LIN {X 0,Y 720.771,Z 351.039,A -85,B 0,C 180,E1 33793.667,E2 33793.667} C_VEL
LIN {X 0,Y 724.023,Z 364.249,A -85,B 0,C 180,E1 33793.246,E2 33793.246} C_VEL
LIN {X 0,Y 722.637,Z 576.137,A -85,B 0,C 180,E1 33790.575,E2 33790.575} C_VEL
LIN {X 0,Y 721.291,Z 800.134,A -85,B 0,C 180,E1 33787.845,E2 33787.845} C_VEL
LIN {X 0,Y 720.97,Z 835.449,A -85,B 0,C 180,E1 33787.381,E2 33787.381} C_VEL
LIN {X 0,Y 720.477,Z 862.842,A -85,B 0,C 180,E1 33786.854,E2 33786.854} C_VEL
LIN {X 0,Y 719.962,Z 888.338,A -85,B 0,C 180,E1 33786.211,E2 33786.211} C_VEL
LIN {X 0,Y 719.265,Z 916.706,A -85,B 0,C 180,E1 33785.311,E2 33785.311} C_VEL
LIN {X 0,Y 718.599,Z 939.502,A -85,B 0,C 180,E1 33784.444,E2 33784.444} C_VEL
LIN {X 0,Y 717.941,Z 960.707,A -85,B 0,C 180,E1 33783.518,E2 33783.518} C_VEL
LIN {X 0,Y 717.25,Z 982.995,A -85,B 0,C 180,E1 33782.412,E2 33782.412} C_VEL
LIN {X 0,Y 716.464,Z 1007.893,A -85,B 0,C 180,E1 33780.994,E2 33780.994} C_VEL
LIN {X 0,Y 715.787,Z 1027.578,A -85,B 0,C 180,E1 33779.728,E2 33779.728} C_VEL
LIN {X 0,Y 715.19,Z 1045.813,A -85,B 0,C 180,E1 33778.431,E2 33778.431} C_VEL
LIN {X 0,Y 714.548,Z 1067.22,A -85,B 0,C 180,E1 33776.735,E2 33776.735} C_VEL
LIN {X 0,Y 713.971,Z 1085.454,A -85,B 0,C 180,E1 33775.108,E2 33775.108} C_VEL
LIN {X 0,Y 713.51,Z 1101.397,A -85,B 0,C 180,E1 33773.539,E2 33773.539} C_VEL
LIN {X 0,Y 713.048,Z 1120.128,A -85,B 0,C 180,E1 33771.468,E2 33771.468} C_VEL
LIN {X 0,Y 712.741,Z 1134.092,A -85,B 0,C 180,E1 33769.723,E2 33769.723} C_VEL
LIN {X 0,Y 712.497,Z 1146.006,A -85,B 0,C 180,E1 33768.067,E2 33768.067} C_VEL
LIN {X 0,Y 712.28,Z 1158.901,A -85,B 0,C 180,E1 33766.054,E2 33766.054} C_VEL
LIN {X 0,Y 712.124,Z 1170.245,A -85,B 0,C 180,E1 33763.975,E2 33763.975} C_VEL
LIN {X 0,Y 712.027,Z 1178.433,A -85,B 0,C 180,E1 33762.242,E2 33762.242} C_VEL
LIN {X 0,Y 711.98,Z 1186.134,A -85,B 0,C 180,E1 33760.355,E2 33760.355} C_VEL
LIN {X 0,Y 711.935,Z 1193.355,A -85,B 0,C 180,E1 33758.155,E2 33758.155} C_VEL
LIN {X 0,Y 711.916,Z 1198.765,A -85,B 0,C 180,E1 33755.966,E2 33755.966} C_VEL
LIN {X 0,Y 711.907,Z 1202.382,A -85,B 0,C 180,E1 33753.866,E2 33753.866} C_VEL
LIN {X 0,Y 711.909,Z 1204.549,A -85,B 0,C 180,E1 33751.61,E2 33751.61} C_VEL
LIN {X 0,Y 711.89,Z 1204.872,A -85,B 0,C 180,E1 33749.517,E2 33749.517} C_VEL
LIN {X 0,Y 711.907,Z 1203.967,A -85,B 0,C 180,E1 33747.585,E2 33747.585} C_VEL
LIN {X 0,Y 711.908,Z 1201.303,A -85,B 0,C 180,E1 33745.408,E2 33745.408} C_VEL
LIN {X 0,Y 711.919,Z 1197.152,A -85,B 0,C 180,E1 33743.306,E2 33743.306} C_VEL
LIN {X 0,Y 711.945,Z 1191.397,A -85,B 0,C 180,E1 33741.195,E2 33741.195} C_VEL
LIN {X 0,Y 711.977,Z 1183.958,A -85,B 0,C 180,E1 33739.071,E2 33739.071} C_VEL
LIN {X 0,Y 712.09,Z 1173.94,A -85,B 0,C 180,E1 33736.769,E2 33736.769} C_VEL
LIN {X 0,Y 712.178,Z 1164.531,A -85,B 0,C 180,E1 33734.946,E2 33734.946} C_VEL
LIN {X 0,Y 712.341,Z 1154.745,A -85,B 0,C 180,E1 33733.277,E2 33733.277} C_VEL
LIN {X 0,Y 712.542,Z 1143.678,A -85,B 0,C 180,E1 33731.595,E2 33731.595} C_VEL
LIN {X 0,Y 712.858,Z 1129.296,A -85,B 0,C 180,E1 33729.644,E2 33729.644} C_VEL
LIN {X 0,Y 713.224,Z 1112.625,A -85,B 0,C 180,E1 33727.672,E2 33727.672} C_VEL
LIN {X 0,Y 713.611,Z 1097.983,A -85,B 0,C 180,E1 33726.114,E2 33726.114} C_VEL
LIN {X 0,Y 714.174,Z 1079.334,A -85,B 0,C 180,E1 33724.317,E2 33724.317} C_VEL
LIN {X 0,Y 714.745,Z 1059.887,A -85,B 0,C 180,E1 33722.665,E2 33722.665} C_VEL
LIN {X 0,Y 715.326,Z 1042.24,A -85,B 0,C 180,E1 33721.306,E2 33721.306} C_VEL
LIN {X 0,Y 716.075,Z 1020.251,A -85,B 0,C 180,E1 33719.777,E2 33719.777} C_VEL
LIN {X 0,Y 716.773,Z 997.046,A -85,B 0,C 180,E1 33718.366,E2 33718.366} C_VEL
LIN {X 0,Y 717.451,Z 976.762,A -85,B 0,C 180,E1 33717.267,E2 33717.267} C_VEL
LIN {X 0,Y 718.191,Z 954.383,A -85,B 0,C 180,E1 33716.192,E2 33716.192} C_VEL
LIN {X 0,Y 718.939,Z 927.69,A -85,B 0,C 180,E1 33715.09,E2 33715.09} C_VEL
LIN {X 0,Y 719.505,Z 905.6,A -85,B 0,C 180,E1 33714.317,E2 33714.317} C_VEL
LIN {X 0,Y 720.071,Z 882.549,A -85,B 0,C 180,E1 33713.63,E2 33713.63} C_VEL
LIN {X 0,Y 720.646,Z 855.599,A -85,B 0,C 180,E1 33712.99,E2 33712.99} C_VEL
LIN {X 0,Y 721.041,Z 828.402,A -85,B 0,C 180,E1 33712.512,E2 33712.512} C_VEL
LIN {X 0,Y 722.489,Z 599.337,A -85,B 0,C 180,E1 33709.712,E2 33709.712} C_VEL
LIN {X 0,Y 723.84,Z 391.194,A -85,B 0,C 180,E1 33707.099,E2 33707.099} C_VEL
LIN {X 0,Y 723.859,Z 362.91,A -85,B 0,C 180,E1 33706.724,E2 33706.724} C_VEL
LIN {X 0,Y 720.673,Z 350.184,A -85,B 0,C 180,E1 33706.291,E2 33706.291} C_VEL
LIN {X 0,Y 720.959,Z 334.838,A -85,B 0,C 180,E1 33705.242,E2 33705.242} C_VEL
LIN {X 0,Y 713.885,Z 319.445,A -85,B 0,C 180,E1 33703.56,E2 33703.56} C_VEL
LIN {X 0,Y 712.33,Z 316.032,A -85,B 0,C 180,E1 33703.177,E2 33703.177} C_VEL
LIN {X 0,Y 712.25,Z 315.511,A -85,B 0,C 180,E1 33703.116,E2 33703.116} C_VEL
LIN {X 0,Y 712.269,Z 315.495,A -85,B 0,C 180,E1 33700.213,E2 33700.213} C_VEL
LIN {X 0,Y 712.243,Z 315.502,A -85,B 0,C 180,E1 33697.335,E2 33697.335} C_VEL
LIN {X 0,Y 712.278,Z 315.499,A -85,B 0,C 180,E1 33694.453,E2 33694.453} C_VEL
LIN {X 0,Y 712.252,Z 315.506,A -85,B 0,C 180,E1 33691.388,E2 33691.388} C_VEL
LIN {X 0,Y 712.258,Z 315.499,A -85,B 0,C 180,E1 33688.506,E2 33688.506} C_VEL
LIN {X 0,Y 712.255,Z 315.499,A -85,B 0,C 180,E1 33685.352,E2 33685.352} C_VEL
LIN {X 0,Y 712.24,Z 315.504,A -85,B 0,C 180,E1 33682.525,E2 33682.525} C_VEL
LIN {X 0,Y 712.279,Z 315.497,A -85,B 0,C 180,E1 33679.518,E2 33679.518} C_VEL
LIN {X 0,Y 712.225,Z 315.505,A -85,B 0,C 180,E1 33676.726,E2 33676.726} C_VEL
LIN {X 0,Y 712.27,Z 315.492,A -85,B 0,C 180,E1 33673.973,E2 33673.973} C_VEL
LIN {X 0,Y 712.235,Z 315.505,A -85,B 0,C 180,E1 33670.925,E2 33670.925} C_VEL
LIN {X 0,Y 712.225,Z 315.498,A -85,B 0,C 180,E1 33668.226,E2 33668.226} C_VEL
LIN {X 0,Y 712.281,Z 315.51,A -85,B 0,C 180,E1 33665.316,E2 33665.316} C_VEL
LIN {X 0,Y 712.213,Z 315.501,A -85,B 0,C 180,E1 33662.494,E2 33662.494} C_VEL
LIN {X 0,Y 712.227,Z 315.506,A -85,B 0,C 180,E1 33659.92,E2 33659.92} C_VEL
LIN {X 0,Y 712.251,Z 315.499,A -85,B 0,C 180,E1 33656.861,E2 33656.861} C_VEL
LIN {X 0,Y 712.205,Z 315.509,A -85,B 0,C 180,E1 33654.198,E2 33654.198} C_VEL
LIN {X 0,Y 712.231,Z 315.5,A -85,B 0,C 180,E1 33651.605,E2 33651.605} C_VEL
LIN {X 0,Y 712.22,Z 315.511,A -85,B 0,C 180,E1 33648.49,E2 33648.49} C_VEL
LIN {X 0,Y 712.196,Z 315.502,A -85,B 0,C 180,E1 33645.953,E2 33645.953} C_VEL
LIN {X 0,Y 712.231,Z 315.503,A -85,B 0,C 180,E1 33643.358,E2 33643.358} C_VEL
LIN {X 0,Y 712.28,Z 315.503,A -85,B 0,C 180,E1 33640.816,E2 33640.816} C_VEL
LIN {X 0,Y 711.26,Z 315.62,A -85,B 0,C 180,E1 33640.197,E2 33640.197} C_VEL
LIN {X 0,Y 704.805,Z 316.435,A -85,B 0,C 180,E1 33638.461,E2 33638.461} C_VEL
LIN {X 0,Y 704.255,Z 316.499,A -85,B 0,C 180,E1 33638.01,E2 33638.01} C_VEL
LIN {X 0,Y 704.249,Z 316.497,A -85,B 0,C 180,E1 33635.596,E2 33635.596} C_VEL
LIN {X 0,Y 704.329,Z 316.492,A -85,B 0,C 180,E1 33632.798,E2 33632.798} C_VEL
LIN {X 0,Y 704.251,Z 316.488,A -85,B 0,C 180,E1 33629.921,E2 33629.921} C_VEL
LIN {X 0,Y 704.239,Z 316.502,A -85,B 0,C 180,E1 33627.495,E2 33627.495} C_VEL
LIN {X 0,Y 704.264,Z 316.488,A -85,B 0,C 180,E1 33624.999,E2 33624.999} C_VEL
LIN {X 0,Y 704.252,Z 316.49,A -85,B 0,C 180,E1 33621.858,E2 33621.858} C_VEL
LIN {X 0,Y 704.231,Z 316.505,A -85,B 0,C 180,E1 33619.427,E2 33619.427} C_VEL
LIN {X 0,Y 704.241,Z 316.504,A -85,B 0,C 180,E1 33617.038,E2 33617.038} C_VEL
LIN {X 0,Y 704.252,Z 316.642,A -85,B 0,C 180,E1 33615.256,E2 33615.256} C_VEL
LIN {X 0,Y 705.594,Z 320.045,A -85,B 0,C 180,E1 33614.883,E2 33614.883} C_VEL
LIN {X 0,Y 706.502,Z 321.785,A -85,B 0,C 180,E1 33614.727,E2 33614.727} C_VEL
LIN {X 0,Y 718.08,Z 339.407,A -85,B 0,C 180,E1 33613.579,E2 33613.579} C_VEL
LIN {X 0,Y 716.627,Z 536.634,A -85,B 0,C 180,E1 33611.066,E2 33611.066} C_VEL
LIN {X 0,Y 715.015,Z 763.363,A -85,B 0,C 180,E1 33608.276,E2 33608.276} C_VEL
LIN {X 0,Y 714.605,Z 804.25,A -85,B 0,C 180,E1 33607.747,E2 33607.747} C_VEL
LIN {X 0,Y 714.056,Z 831.612,A -85,B 0,C 180,E1 33607.225,E2 33607.225} C_VEL
LIN {X 0,Y 713.456,Z 856.532,A -85,B 0,C 180,E1 33606.602,E2 33606.602} C_VEL
LIN {X 0,Y 712.726,Z 883.752,A -85,B 0,C 180,E1 33605.753,E2 33605.753} C_VEL
LIN {X 0,Y 711.881,Z 908.474,A -85,B 0,C 180,E1 33604.816,E2 33604.816} C_VEL
LIN {X 0,Y 711.111,Z 929.791,A -85,B 0,C 180,E1 33603.883,E2 33603.883} C_VEL
LIN {X 0,Y 710.333,Z 950.383,A -85,B 0,C 180,E1 33602.862,E2 33602.862} C_VEL
LIN {X 0,Y 709.442,Z 974.728,A -85,B 0,C 180,E1 33601.494,E2 33601.494} C_VEL
LIN {X 0,Y 708.6,Z 996.129,A -85,B 0,C 180,E1 33600.118,E2 33600.118} C_VEL
LIN {X 0,Y 707.868,Z 1014.676,A -85,B 0,C 180,E1 33598.794,E2 33598.794} C_VEL
LIN {X 0,Y 707.09,Z 1035.698,A -85,B 0,C 180,E1 33597.131,E2 33597.131} C_VEL
LIN {X 0,Y 706.407,Z 1054.988,A -85,B 0,C 180,E1 33595.396,E2 33595.396} C_VEL
LIN {X 0,Y 705.839,Z 1071.299,A -85,B 0,C 180,E1 33593.776,E2 33593.776} C_VEL
LIN {X 0,Y 705.294,Z 1089.764,A -85,B 0,C 180,E1 33591.716,E2 33591.716} C_VEL
LIN {X 0,Y 704.924,Z 1103.476,A -85,B 0,C 180,E1 33589.988,E2 33589.988} C_VEL
LIN {X 0,Y 704.625,Z 1115.703,A -85,B 0,C 180,E1 33588.276,E2 33588.276} C_VEL
LIN {X 0,Y 704.363,Z 1128.113,A -85,B 0,C 180,E1 33586.324,E2 33586.324} C_VEL
LIN {X 0,Y 704.168,Z 1140.163,A -85,B 0,C 180,E1 33584.108,E2 33584.108} C_VEL
LIN {X 0,Y 704.054,Z 1148.655,A -85,B 0,C 180,E1 33582.286,E2 33582.286} C_VEL
LIN {X 0,Y 703.993,Z 1156.268,A -85,B 0,C 180,E1 33580.392,E2 33580.392} C_VEL
LIN {X 0,Y 703.948,Z 1163.465,A -85,B 0,C 180,E1 33578.166,E2 33578.166} C_VEL
LIN {X 0,Y 703.923,Z 1168.842,A -85,B 0,C 180,E1 33575.952,E2 33575.952} C_VEL
LIN {X 0,Y 703.911,Z 1172.427,A -85,B 0,C 180,E1 33573.828,E2 33573.828} C_VEL
LIN {X 0,Y 703.907,Z 1174.519,A -85,B 0,C 180,E1 33571.628,E2 33571.628} C_VEL
LIN {X 0,Y 703.89,Z 1174.884,A -85,B 0,C 180,E1 33569.512,E2 33569.512} C_VEL
LIN {X 0,Y 703.905,Z 1173.934,A -85,B 0,C 180,E1 33567.476,E2 33567.476} C_VEL
LIN {X 0,Y 703.909,Z 1171.247,A -85,B 0,C 180,E1 33565.274,E2 33565.274} C_VEL
LIN {X 0,Y 703.919,Z 1167.064,A -85,B 0,C 180,E1 33563.147,E2 33563.147} C_VEL
LIN {X 0,Y 703.951,Z 1161.278,A -85,B 0,C 180,E1 33561.011,E2 33561.011} C_VEL
LIN {X 0,Y 704.003,Z 1153.813,A -85,B 0,C 180,E1 33558.863,E2 33558.863} C_VEL
LIN {X 0,Y 704.126,Z 1143.751,A -85,B 0,C 180,E1 33556.533,E2 33556.533} C_VEL
LIN {X 0,Y 704.243,Z 1134.314,A -85,B 0,C 180,E1 33554.688,E2 33554.688} C_VEL
LIN {X 0,Y 704.447,Z 1124.499,A -85,B 0,C 180,E1 33552.999,E2 33552.999} C_VEL
LIN {X 0,Y 704.706,Z 1112.819,A -85,B 0,C 180,E1 33551.212,E2 33551.212} C_VEL
LIN {X 0,Y 705.097,Z 1096.881,A -85,B 0,C 180,E1 33549.063,E2 33549.063} C_VEL
LIN {X 0,Y 705.498,Z 1082.171,A -85,B 0,C 180,E1 33547.318,E2 33547.318} C_VEL
LIN {X 0,Y 705.976,Z 1067.563,A -85,B 0,C 180,E1 33545.75,E2 33545.75} C_VEL
LIN {X 0,Y 706.596,Z 1049.287,A -85,B 0,C 180,E1 33543.972,E2 33543.972} C_VEL
LIN {X 0,Y 707.315,Z 1029.605,A -85,B 0,C 180,E1 33542.285,E2 33542.285} C_VEL
LIN {X 0,Y 707.977,Z 1012.225,A -85,B 0,C 180,E1 33540.934,E2 33540.934} C_VEL
LIN {X 0,Y 708.85,Z 989.911,A -85,B 0,C 180,E1 33539.368,E2 33539.368} C_VEL
LIN {X 0,Y 709.707,Z 967.008,A -85,B 0,C 180,E1 33537.966,E2 33537.966} C_VEL
LIN {X 0,Y 710.487,Z 946.818,A -85,B 0,C 180,E1 33536.863,E2 33536.863} C_VEL
LIN {X 0,Y 711.289,Z 925.649,A -85,B 0,C 180,E1 33535.835,E2 33535.835} C_VEL
LIN {X 0,Y 712.17,Z 900.127,A -85,B 0,C 180,E1 33534.758,E2 33534.758} C_VEL
LIN {X 0,Y 712.878,Z 875.711,A -85,B 0,C 180,E1 33533.892,E2 33533.892} C_VEL
LIN {X 0,Y 713.545,Z 852.788,A -85,B 0,C 180,E1 33533.205,E2 33533.205} C_VEL
LIN {X 0,Y 714.206,Z 825.892,A -85,B 0,C 180,E1 33532.561,E2 33532.561} C_VEL
LIN {X 0,Y 714.674,Z 798.761,A -85,B 0,C 180,E1 33532.08,E2 33532.08} C_VEL
LIN {X 0,Y 716.381,Z 570.178,A -85,B 0,C 180,E1 33529.262,E2 33529.262} C_VEL
LIN {X 0,Y 717.934,Z 362.47,A -85,B 0,C 180,E1 33526.632,E2 33526.632} C_VEL
LIN {X 0,Y 717.96,Z 338.909,A -85,B 0,C 180,E1 33526.316,E2 33526.316} C_VEL
LIN {X 0,Y 707.614,Z 323.566,A -85,B 0,C 180,E1 33525.297,E2 33525.297} C_VEL
LIN {X 0,Y 705.936,Z 320.494,A -85,B 0,C 180,E1 33525.089,E2 33525.089} C_VEL
LIN {X 0,Y 704.379,Z 317.274,A -85,B 0,C 180,E1 33524.714,E2 33524.714} C_VEL
LIN {X 0,Y 704.245,Z 316.508,A -85,B 0,C 180,E1 33524.609,E2 33524.609} C_VEL
LIN {X 0,Y 704.277,Z 316.501,A -85,B 0,C 180,E1 33522.055,E2 33522.055} C_VEL
LIN {X 0,Y 704.256,Z 316.504,A -85,B 0,C 180,E1 33518.974,E2 33518.974} C_VEL
LIN {X 0,Y 704.234,Z 316.504,A -85,B 0,C 180,E1 33516.506,E2 33516.506} C_VEL
LIN {X 0,Y 704.241,Z 316.49,A -85,B 0,C 180,E1 33514.113,E2 33514.113} C_VEL
LIN {X 0,Y 704.294,Z 316.489,A -85,B 0,C 180,E1 33511.124,E2 33511.124} C_VEL
LIN {X 0,Y 704.239,Z 316.502,A -85,B 0,C 180,E1 33508.494,E2 33508.494} C_VEL
LIN {X 0,Y 704.24,Z 316.495,A -85,B 0,C 180,E1 33506.113,E2 33506.113} C_VEL
LIN {X 0,Y 704.329,Z 316.499,A -85,B 0,C 180,E1 33503.296,E2 33503.296} C_VEL
LIN {X 0,Y 704.254,Z 316.485,A -85,B 0,C 180,E1 33500.442,E2 33500.442} C_VEL
LIN {X 0,Y 704.251,Z 316.499,A -85,B 0,C 180,E1 33497.968,E2 33497.968} C_VEL
LIN {X 0,Y 704.319,Z 316.487,A -85,B 0,C 180,E1 33495.227,E2 33495.227} C_VEL
LIN {X 0,Y 704.268,Z 316.498,A -85,B 0,C 180,E1 33492.296,E2 33492.296} C_VEL
LIN {X 0,Y 704.257,Z 316.493,A -85,B 0,C 180,E1 33489.81,E2 33489.81} C_VEL
LIN {X 0,Y 704.32,Z 316.492,A -85,B 0,C 180,E1 33487.095,E2 33487.095} C_VEL
LIN {X 0,Y 704.279,Z 316.49,A -85,B 0,C 180,E1 33484.152,E2 33484.152} C_VEL
LIN {X 0,Y 704.269,Z 316.489,A -85,B 0,C 180,E1 33481.546,E2 33481.546} C_VEL
LIN {X 0,Y 704.344,Z 316.492,A -85,B 0,C 180,E1 33478.698,E2 33478.698} C_VEL
LIN {X 0,Y 704.276,Z 316.487,A -85,B 0,C 180,E1 33475.766,E2 33475.766} C_VEL
LIN {X 0,Y 704.29,Z 316.499,A -85,B 0,C 180,E1 33473.151,E2 33473.151} C_VEL
LIN {X 0,Y 704.326,Z 316.485,A -85,B 0,C 180,E1 33470.109,E2 33470.109} C_VEL
LIN {X 0,Y 704.28,Z 316.496,A -85,B 0,C 180,E1 33467.371,E2 33467.371} C_VEL
LIN {X 0,Y 704.343,Z 316.484,A -85,B 0,C 180,E1 33464.521,E2 33464.521} C_VEL
LIN {X 0,Y 704.294,Z 316.493,A -85,B 0,C 180,E1 33461.543,E2 33461.543} C_VEL
LIN {X 0,Y 704.308,Z 316.486,A -85,B 0,C 180,E1 33458.776,E2 33458.776} C_VEL
LIN {X 0,Y 704.326,Z 316.483,A -85,B 0,C 180,E1 33455.688,E2 33455.688} C_VEL
LIN {X 0,Y 704.297,Z 316.495,A -85,B 0,C 180,E1 33452.888,E2 33452.888} C_VEL
LIN {X 0,Y 704.338,Z 316.485,A -85,B 0,C 180,E1 33449.99,E2 33449.99} C_VEL
LIN {X 0,Y 704.3,Z 316.493,A -85,B 0,C 180,E1 33447.061,E2 33447.061} C_VEL
LIN {X 0,Y 704.34,Z 316.498,A -85,B 0,C 180,E1 33444.152,E2 33444.152} C_VEL
LIN {X 0,Y 704.317,Z 316.495,A -85,B 0,C 180,E1 33441.135,E2 33441.135} C_VEL
LIN {X 0,Y 704.339,Z 316.499,A -85,B 0,C 180,E1 33438.147,E2 33438.147} C_VEL
LIN {X 0,Y 704.354,Z 316.627,A -85,B 0,C 180,E1 33437.474,E2 33437.474} C_VEL
LIN {X 0,Y 705.691,Z 320.07,A -85,B 0,C 180,E1 33437.097,E2 33437.097} C_VEL
LIN {X 0,Y 712.541,Z 334.723,A -85,B 0,C 180,E1 33435.441,E2 33435.441} C_VEL
LIN {X 0,Y 714.569,Z 339.653,A -85,B 0,C 180,E1 33434.924,E2 33434.924} C_VEL
LIN {X 0,Y 714.39,Z 351.16,A -85,B 0,C 180,E1 33434.156,E2 33434.156} C_VEL
LIN {X 0,Y 718.167,Z 366.394,A -85,B 0,C 180,E1 33433.658,E2 33433.658} C_VEL
LIN {X 0,Y 716.542,Z 577.372,A -85,B 0,C 180,E1 33430.977,E2 33430.977} C_VEL
LIN {X 0,Y 714.958,Z 801.305,A -85,B 0,C 180,E1 33428.225,E2 33428.225} C_VEL
LIN {X 0,Y 714.581,Z 835.878,A -85,B 0,C 180,E1 33427.766,E2 33427.766} C_VEL
LIN {X 0,Y 714.012,Z 863.03,A -85,B 0,C 180,E1 33427.239,E2 33427.239} C_VEL
LIN {X 0,Y 713.419,Z 888.317,A -85,B 0,C 180,E1 33426.597,E2 33426.597} C_VEL
LIN {X 0,Y 712.6,Z 916.851,A -85,B 0,C 180,E1 33425.686,E2 33425.686} C_VEL
LIN {X 0,Y 711.838,Z 939.505,A -85,B 0,C 180,E1 33424.818,E2 33424.818} C_VEL
LIN {X 0,Y 711.114,Z 959.717,A -85,B 0,C 180,E1 33423.931,E2 33423.931} C_VEL
LIN {X 0,Y 710.335,Z 980.327,A -85,B 0,C 180,E1 33422.91,E2 33422.91} C_VEL
LIN {X 0,Y 709.435,Z 1004.952,A -85,B 0,C 180,E1 33421.525,E2 33421.525} C_VEL
LIN {X 0,Y 708.563,Z 1026.865,A -85,B 0,C 180,E1 33420.113,E2 33420.113} C_VEL
LIN {X 0,Y 707.854,Z 1045.266,A -85,B 0,C 180,E1 33418.794,E2 33418.794} C_VEL
LIN {X 0,Y 707.076,Z 1066.205,A -85,B 0,C 180,E1 33417.132,E2 33417.132} C_VEL
LIN {X 0,Y 706.405,Z 1085.046,A -85,B 0,C 180,E1 33415.435,E2 33415.435} C_VEL
LIN {X 0,Y 705.831,Z 1101.399,A -85,B 0,C 180,E1 33413.811,E2 33413.811} C_VEL
LIN {X 0,Y 705.276,Z 1120.13,A -85,B 0,C 180,E1 33411.716,E2 33411.716} C_VEL
LIN {X 0,Y 704.918,Z 1133.811,A -85,B 0,C 180,E1 33409.989,E2 33409.989} C_VEL
LIN {X 0,Y 704.607,Z 1146.59,A -85,B 0,C 180,E1 33408.191,E2 33408.191} C_VEL
LIN {X 0,Y 704.335,Z 1160.068,A -85,B 0,C 180,E1 33406.036,E2 33406.036} C_VEL
LIN {X 0,Y 704.164,Z 1170.657,A -85,B 0,C 180,E1 33404.052,E2 33404.052} C_VEL
LIN {X 0,Y 704.053,Z 1178.792,A -85,B 0,C 180,E1 33402.299,E2 33402.299} C_VEL
LIN {X 0,Y 703.99,Z 1186.427,A -85,B 0,C 180,E1 33400.392,E2 33400.392} C_VEL
LIN {X 0,Y 703.94,Z 1193.595,A -85,B 0,C 180,E1 33398.166,E2 33398.166} C_VEL
LIN {X 0,Y 703.918,Z 1198.937,A -85,B 0,C 180,E1 33395.952,E2 33395.952} C_VEL
LIN {X 0,Y 703.908,Z 1202.484,A -85,B 0,C 180,E1 33393.828,E2 33393.828} C_VEL
LIN {X 0,Y 703.908,Z 1204.549,A -85,B 0,C 180,E1 33391.628,E2 33391.628} C_VEL
LIN {X 0,Y 703.89,Z 1204.872,A -85,B 0,C 180,E1 33389.512,E2 33389.512} C_VEL
LIN {X 0,Y 703.907,Z 1203.964,A -85,B 0,C 180,E1 33387.558,E2 33387.558} C_VEL
LIN {X 0,Y 703.909,Z 1201.428,A -85,B 0,C 180,E1 33385.438,E2 33385.438} C_VEL
LIN {X 0,Y 703.921,Z 1197.348,A -85,B 0,C 180,E1 33383.311,E2 33383.311} C_VEL
LIN {X 0,Y 703.949,Z 1191.394,A -85,B 0,C 180,E1 33381.094,E2 33381.094} C_VEL
LIN {X 0,Y 703.992,Z 1184.277,A -85,B 0,C 180,E1 33379.029,E2 33379.029} C_VEL
LIN {X 0,Y 704.128,Z 1173.941,A -85,B 0,C 180,E1 33376.617,E2 33376.617} C_VEL
LIN {X 0,Y 704.237,Z 1164.533,A -85,B 0,C 180,E1 33374.772,E2 33374.772} C_VEL
LIN {X 0,Y 704.437,Z 1154.7,A -85,B 0,C 180,E1 33373.076,E2 33373.076} C_VEL
LIN {X 0,Y 704.667,Z 1143.68,A -85,B 0,C 180,E1 33371.382,E2 33371.382} C_VEL
LIN {X 0,Y 705.06,Z 1128.62,A -85,B 0,C 180,E1 33369.322,E2 33369.322} C_VEL
LIN {X 0,Y 705.487,Z 1112.627,A -85,B 0,C 180,E1 33367.414,E2 33367.414} C_VEL
LIN {X 0,Y 705.974,Z 1097.61,A -85,B 0,C 180,E1 33365.8,E2 33365.8} C_VEL
LIN {X 0,Y 706.607,Z 1078.762,A -85,B 0,C 180,E1 33363.97,E2 33363.97} C_VEL
LIN {X 0,Y 707.314,Z 1059.614,A -85,B 0,C 180,E1 33362.331,E2 33362.331} C_VEL
LIN {X 0,Y 707.955,Z 1042.846,A -85,B 0,C 180,E1 33361.025,E2 33361.025} C_VEL
LIN {X 0,Y 708.73,Z 1022.922,A -85,B 0,C 180,E1 33359.618,E2 33359.618} C_VEL
LIN {X 0,Y 709.633,Z 998.654,A -85,B 0,C 180,E1 33358.105,E2 33358.105} C_VEL
LIN {X 0,Y 710.413,Z 978.546,A -85,B 0,C 180,E1 33356.998,E2 33356.998} C_VEL
LIN {X 0,Y 711.154,Z 958.824,A -85,B 0,C 180,E1 33356.027,E2 33356.027} C_VEL
LIN {X 0,Y 711.932,Z 937.251,A -85,B 0,C 180,E1 33355.089,E2 33355.089} C_VEL
LIN {X 0,Y 712.777,Z 911.467,A -85,B 0,C 180,E1 33354.126,E2 33354.126} C_VEL
LIN {X 0,Y 713.471,Z 885.657,A -85,B 0,C 180,E1 33353.329,E2 33353.329} C_VEL
LIN {X 0,Y 714.088,Z 860.466,A -85,B 0,C 180,E1 33352.705,E2 33352.705} C_VEL
LIN {X 0,Y 714.616,Z 832.883,A -85,B 0,C 180,E1 33352.187,E2 33352.187} C_VEL
LIN {X 0,Y 715.061,Z 786.137,A -85,B 0,C 180,E1 33351.591,E2 33351.591} C_VEL
LIN {X 0,Y 716.677,Z 560.284,A -85,B 0,C 180,E1 33348.809,E2 33348.809} C_VEL
LIN {X 0,Y 718.112,Z 365.493,A -85,B 0,C 180,E1 33346.326,E2 33346.326} C_VEL
LIN {X 0,Y 714.26,Z 350.268,A -85,B 0,C 180,E1 33345.803,E2 33345.803} C_VEL
LIN {X 0,Y 714.571,Z 339.143,A -85,B 0,C 180,E1 33345.04,E2 33345.04} C_VEL
LIN {X 0,Y 707.611,Z 324.147,A -85,B 0,C 180,E1 33343.373,E2 33343.373} C_VEL
LIN {X 0,Y 705.51,Z 319.793,A -85,B 0,C 180,E1 33342.866,E2 33342.866} C_VEL
LIN {X 0,Y 704.337,Z 316.498,A -85,B 0,C 180,E1 33342.512,E2 33342.512} C_VEL
LIN {X 0,Y 704.314,Z 316.501,A -85,B 0,C 180,E1 33339.495,E2 33339.495} C_VEL
LIN {X 0,Y 704.337,Z 316.487,A -85,B 0,C 180,E1 33336.537,E2 33336.537} C_VEL
LIN {X 0,Y 704.313,Z 316.49,A -85,B 0,C 180,E1 33333.424,E2 33333.424} C_VEL
LIN {X 0,Y 704.328,Z 316.487,A -85,B 0,C 180,E1 33330.493,E2 33330.493} C_VEL
LIN {X 0,Y 704.318,Z 316.498,A -85,B 0,C 180,E1 33327.385,E2 33327.385} C_VEL
LIN {X 0,Y 704.309,Z 316.484,A -85,B 0,C 180,E1 33324.491,E2 33324.491} C_VEL
LIN {X 0,Y 704.33,Z 316.488,A -85,B 0,C 180,E1 33321.398,E2 33321.398} C_VEL
LIN {X 0,Y 704.292,Z 316.493,A -85,B 0,C 180,E1 33318.543,E2 33318.543} C_VEL
LIN {X 0,Y 704.342,Z 316.488,A -85,B 0,C 180,E1 33315.648,E2 33315.648} C_VEL
LIN {X 0,Y 704.287,Z 316.497,A -85,B 0,C 180,E1 33312.758,E2 33312.758} C_VEL
LIN {X 0,Y 704.317,Z 316.487,A -85,B 0,C 180,E1 33309.974,E2 33309.974} C_VEL
LIN {X 0,Y 704.303,Z 316.5,A -85,B 0,C 180,E1 33306.931,E2 33306.931} C_VEL
LIN {X 0,Y 704.279,Z 316.489,A -85,B 0,C 180,E1 33304.234,E2 33304.234} C_VEL
LIN {X 0,Y 704.345,Z 316.489,A -85,B 0,C 180,E1 33301.302,E2 33301.302} C_VEL
LIN {X 0,Y 704.275,Z 316.491,A -85,B 0,C 180,E1 33298.454,E2 33298.454} C_VEL
LIN {X 0,Y 704.281,Z 316.488,A -85,B 0,C 180,E1 33295.848,E2 33295.848} C_VEL
LIN {X 0,Y 704.316,Z 316.493,A -85,B 0,C 180,E1 33292.823,E2 33292.823} C_VEL
LIN {X 0,Y 704.263,Z 316.491,A -85,B 0,C 180,E1 33290.158,E2 33290.158} C_VEL
LIN {X 0,Y 704.279,Z 316.497,A -85,B 0,C 180,E1 33287.619,E2 33287.619} C_VEL
LIN {X 0,Y 704.292,Z 316.492,A -85,B 0,C 180,E1 33284.52,E2 33284.52} C_VEL
LIN {X 0,Y 704.255,Z 316.499,A -85,B 0,C 180,E1 33281.97,E2 33281.97} C_VEL
LIN {X 0,Y 704.264,Z 316.485,A -85,B 0,C 180,E1 33279.471,E2 33279.471} C_VEL
LIN {X 0,Y 704.255,Z 316.499,A -85,B 0,C 180,E1 33278.01,E2 33278.01} C_VEL
LIN {X 0,Y 703.238,Z 316.628,A -85,B 0,C 180,E1 33277.383,E2 33277.383} C_VEL
LIN {X 0,Y 696.828,Z 317.423,A -85,B 0,C 180,E1 33275.627,E2 33275.627} C_VEL
LIN {X 0,Y 696.343,Z 317.485,A -85,B 0,C 180,E1 33275.171,E2 33275.171} C_VEL
LIN {X 0,Y 696.325,Z 317.491,A -85,B 0,C 180,E1 33272.087,E2 33272.087} C_VEL
LIN {X 0,Y 696.302,Z 317.475,A -85,B 0,C 180,E1 33269.637,E2 33269.637} C_VEL
LIN {X 0,Y 696.321,Z 317.491,A -85,B 0,C 180,E1 33267.126,E2 33267.126} C_VEL
LIN {X 0,Y 696.32,Z 317.494,A -85,B 0,C 180,E1 33263.942,E2 33263.942} C_VEL
LIN {X 0,Y 696.292,Z 317.478,A -85,B 0,C 180,E1 33261.447,E2 33261.447} C_VEL
LIN {X 0,Y 696.308,Z 317.494,A -85,B 0,C 180,E1 33258.985,E2 33258.985} C_VEL
LIN {X 0,Y 696.346,Z 317.495,A -85,B 0,C 180,E1 33255.974,E2 33255.974} C_VEL
LIN {X 0,Y 696.371,Z 317.803,A -85,B 0,C 180,E1 33255.823,E2 33255.823} C_VEL
LIN {X 0,Y 697.895,Z 321.383,A -85,B 0,C 180,E1 33255.438,E2 33255.438} C_VEL
LIN {X 0,Y 701.49,Z 326.53,A -85,B 0,C 180,E1 33255.067,E2 33255.067} C_VEL
LIN {X 0,Y 712.247,Z 343.156,A -85,B 0,C 180,E1 33253.976,E2 33253.976} C_VEL
LIN {X 0,Y 710.567,Z 539.356,A -85,B 0,C 180,E1 33251.458,E2 33251.458} C_VEL
LIN {X 0,Y 708.714,Z 765.576,A -85,B 0,C 180,E1 33248.652,E2 33248.652} C_VEL
LIN {X 0,Y 708.255,Z 804.915,A -85,B 0,C 180,E1 33248.136,E2 33248.136} C_VEL
LIN {X 0,Y 707.62,Z 832.271,A -85,B 0,C 180,E1 33247.606,E2 33247.606} C_VEL
LIN {X 0,Y 706.937,Z 856.943,A -85,B 0,C 180,E1 33246.983,E2 33246.983} C_VEL
LIN {X 0,Y 706.108,Z 883.765,A -85,B 0,C 180,E1 33246.141,E2 33246.141} C_VEL
LIN {X 0,Y 705.151,Z 908.485,A -85,B 0,C 180,E1 33245.197,E2 33245.197} C_VEL
LIN {X 0,Y 704.3,Z 929.261,A -85,B 0,C 180,E1 33244.283,E2 33244.283} C_VEL
LIN {X 0,Y 703.426,Z 949.507,A -85,B 0,C 180,E1 33243.275,E2 33243.275} C_VEL
LIN {X 0,Y 702.397,Z 972.99,A -85,B 0,C 180,E1 33241.958,E2 33241.958} C_VEL
LIN {X 0,Y 701.393,Z 995.625,A -85,B 0,C 180,E1 33240.497,E2 33240.497} C_VEL
LIN {X 0,Y 700.56,Z 1014.141,A -85,B 0,C 180,E1 33239.165,E2 33239.165} C_VEL
LIN {X 0,Y 699.716,Z 1033.482,A -85,B 0,C 180,E1 33237.627,E2 33237.627} C_VEL
LIN {X 0,Y 698.891,Z 1053.297,A -85,B 0,C 180,E1 33235.855,E2 33235.855} C_VEL
LIN {X 0,Y 698.263,Z 1069.266,A -85,B 0,C 180,E1 33234.265,E2 33234.265} C_VEL
LIN {X 0,Y 697.658,Z 1086.03,A -85,B 0,C 180,E1 33232.418,E2 33232.418} C_VEL
LIN {X 0,Y 697.129,Z 1102.193,A -85,B 0,C 180,E1 33230.397,E2 33230.397} C_VEL
LIN {X 0,Y 696.79,Z 1114.544,A -85,B 0,C 180,E1 33228.662,E2 33228.662} C_VEL
LIN {X 0,Y 696.504,Z 1126.043,A -85,B 0,C 180,E1 33226.857,E2 33226.857} C_VEL
LIN {X 0,Y 696.267,Z 1138.389,A -85,B 0,C 180,E1 33224.64,E2 33224.64} C_VEL
LIN {X 0,Y 696.102,Z 1148.244,A -85,B 0,C 180,E1 33222.526,E2 33222.526} C_VEL
LIN {X 0,Y 695.996,Z 1155.965,A -85,B 0,C 180,E1 33220.596,E2 33220.596} C_VEL
LIN {X 0,Y 695.957,Z 1163.223,A -85,B 0,C 180,E1 33218.343,E2 33218.343} C_VEL
LIN {X 0,Y 695.927,Z 1168.672,A -85,B 0,C 180,E1 33216.103,E2 33216.103} C_VEL
LIN {X 0,Y 695.915,Z 1172.318,A -85,B 0,C 180,E1 33213.954,E2 33213.954} C_VEL
LIN {X 0,Y 695.906,Z 1174.463,A -85,B 0,C 180,E1 33211.729,E2 33211.729} C_VEL
LIN {X 0,Y 695.89,Z 1174.884,A -85,B 0,C 180,E1 33209.506,E2 33209.506} C_VEL
LIN {X 0,Y 695.907,Z 1173.999,A -85,B 0,C 180,E1 33207.53,E2 33207.53} C_VEL
LIN {X 0,Y 695.908,Z 1171.496,A -85,B 0,C 180,E1 33205.385,E2 33205.385} C_VEL
LIN {X 0,Y 695.922,Z 1167.454,A -85,B 0,C 180,E1 33203.234,E2 33203.234} C_VEL
LIN {X 0,Y 695.957,Z 1161.528,A -85,B 0,C 180,E1 33200.991,E2 33200.991} C_VEL
LIN {X 0,Y 696.015,Z 1154.336,A -85,B 0,C 180,E1 33198.872,E2 33198.872} C_VEL
LIN {X 0,Y 696.159,Z 1144.155,A -85,B 0,C 180,E1 33196.461,E2 33196.461} C_VEL
LIN {X 0,Y 696.301,Z 1134.778,A -85,B 0,C 180,E1 33194.594,E2 33194.594} C_VEL
LIN {X 0,Y 696.535,Z 1124.497,A -85,B 0,C 180,E1 33192.8,E2 33192.8} C_VEL
LIN {X 0,Y 696.842,Z 1112.817,A -85,B 0,C 180,E1 33190.992,E2 33190.992} C_VEL
LIN {X 0,Y 697.304,Z 1096.874,A -85,B 0,C 180,E1 33188.818,E2 33188.818} C_VEL
LIN {X 0,Y 697.776,Z 1082.243,A -85,B 0,C 180,E1 33187.061,E2 33187.061} C_VEL
LIN {X 0,Y 698.365,Z 1066.705,A -85,B 0,C 180,E1 33185.378,E2 33185.378} C_VEL
LIN {X 0,Y 699.173,Z 1046.349,A -85,B 0,C 180,E1 33183.41,E2 33183.41} C_VEL
LIN {X 0,Y 699.913,Z 1029.044,A -85,B 0,C 180,E1 33181.92,E2 33181.92} C_VEL
LIN {X 0,Y 700.688,Z 1011.093,A -85,B 0,C 180,E1 33180.515,E2 33180.515} C_VEL
LIN {X 0,Y 701.705,Z 988.261,A -85,B 0,C 180,E1 33178.914,E2 33178.914} C_VEL
LIN {X 0,Y 702.664,Z 967.001,A -85,B 0,C 180,E1 33177.606,E2 33177.606} C_VEL
LIN {X 0,Y 703.516,Z 947.591,A -85,B 0,C 180,E1 33176.534,E2 33176.534} C_VEL
LIN {X 0,Y 704.393,Z 927.29,A -85,B 0,C 180,E1 33175.535,E2 33175.535} C_VEL
LIN {X 0,Y 705.424,Z 902.137,A -85,B 0,C 180,E1 33174.45,E2 33174.45} C_VEL
LIN {X 0,Y 706.281,Z 876.183,A -85,B 0,C 180,E1 33173.517,E2 33173.517} C_VEL
LIN {X 0,Y 707.044,Z 853.194,A -85,B 0,C 180,E1 33172.824,E2 33172.824} C_VEL
LIN {X 0,Y 707.777,Z 826.912,A -85,B 0,C 180,E1 33172.186,E2 33172.186} C_VEL
LIN {X 0,Y 708.336,Z 799.401,A -85,B 0,C 180,E1 33171.69,E2 33171.69} C_VEL
LIN {X 0,Y 710.27,Z 574.638,A -85,B 0,C 180,E1 33168.896,E2 33168.896} C_VEL
LIN {X 0,Y 712.082,Z 365.35,A -85,B 0,C 180,E1 33166.225,E2 33166.225} C_VEL
LIN {X 0,Y 712.135,Z 342.734,A -85,B 0,C 180,E1 33165.92,E2 33165.92} C_VEL
LIN {X 0,Y 701.027,Z 326.024,A -85,B 0,C 180,E1 33164.798,E2 33164.798} C_VEL
LIN {X 0,Y 697.409,Z 320.649,A -85,B 0,C 180,E1 33164.4,E2 33164.4} C_VEL
LIN {X 0,Y 696.348,Z 317.495,A -85,B 0,C 180,E1 33164.045,E2 33164.045} C_VEL
LIN {X 0,Y 696.32,Z 317.495,A -85,B 0,C 180,E1 33161.014,E2 33161.014} C_VEL
LIN {X 0,Y 696.297,Z 317.494,A -85,B 0,C 180,E1 33158.553,E2 33158.553} C_VEL
LIN {X 0,Y 696.316,Z 317.493,A -85,B 0,C 180,E1 33156.058,E2 33156.058} C_VEL
LIN {X 0,Y 696.315,Z 317.493,A -85,B 0,C 180,E1 33152.875,E2 33152.875} C_VEL
LIN {X 0,Y 696.295,Z 317.477,A -85,B 0,C 180,E1 33150.459,E2 33150.459} C_VEL
LIN {X 0,Y 696.303,Z 317.491,A -85,B 0,C 180,E1 33148.1,E2 33148.1} C_VEL
LIN {X 0,Y 696.394,Z 317.472,A -85,B 0,C 180,E1 33145.24,E2 33145.24} C_VEL
LIN {X 0,Y 696.308,Z 317.489,A -85,B 0,C 180,E1 33142.367,E2 33142.367} C_VEL
LIN {X 0,Y 696.307,Z 317.473,A -85,B 0,C 180,E1 33139.985,E2 33139.985} C_VEL
LIN {X 0,Y 696.391,Z 317.489,A -85,B 0,C 180,E1 33137.204,E2 33137.204} C_VEL
LIN {X 0,Y 696.319,Z 317.476,A -85,B 0,C 180,E1 33134.248,E2 33134.248} C_VEL
LIN {X 0,Y 696.319,Z 317.489,A -85,B 0,C 180,E1 33131.766,E2 33131.766} C_VEL
LIN {X 0,Y 696.402,Z 317.468,A -85,B 0,C 180,E1 33128.921,E2 33128.921} C_VEL
LIN {X 0,Y 696.327,Z 317.487,A -85,B 0,C 180,E1 33126.017,E2 33126.017} C_VEL
LIN {X 0,Y 696.334,Z 317.481,A -85,B 0,C 180,E1 33123.458,E2 33123.458} C_VEL
LIN {X 0,Y 696.402,Z 317.483,A -85,B 0,C 180,E1 33120.494,E2 33120.494} C_VEL
LIN {X 0,Y 696.332,Z 317.478,A -85,B 0,C 180,E1 33117.696,E2 33117.696} C_VEL
LIN {X 0,Y 696.371,Z 317.479,A -85,B 0,C 180,E1 33114.975,E2 33114.975} C_VEL
LIN {X 0,Y 696.356,Z 317.475,A -85,B 0,C 180,E1 33111.911,E2 33111.911} C_VEL
LIN {X 0,Y 696.342,Z 317.479,A -85,B 0,C 180,E1 33109.241,E2 33109.241} C_VEL
LIN {X 0,Y 696.404,Z 317.471,A -85,B 0,C 180,E1 33106.296,E2 33106.296} C_VEL
LIN {X 0,Y 696.346,Z 317.481,A -85,B 0,C 180,E1 33103.396,E2 33103.396} C_VEL
LIN {X 0,Y 696.395,Z 317.474,A -85,B 0,C 180,E1 33100.542,E2 33100.542} C_VEL
LIN {X 0,Y 696.367,Z 317.483,A -85,B 0,C 180,E1 33097.546,E2 33097.546} C_VEL
LIN {X 0,Y 696.365,Z 317.474,A -85,B 0,C 180,E1 33094.757,E2 33094.757} C_VEL
LIN {X 0,Y 696.399,Z 317.476,A -85,B 0,C 180,E1 33091.656,E2 33091.656} C_VEL
LIN {X 0,Y 696.362,Z 317.483,A -85,B 0,C 180,E1 33088.778,E2 33088.778} C_VEL
LIN {X 0,Y 696.397,Z 317.473,A -85,B 0,C 180,E1 33085.847,E2 33085.847} C_VEL
LIN {X 0,Y 696.365,Z 317.479,A -85,B 0,C 180,E1 33082.97,E2 33082.97} C_VEL
LIN {X 0,Y 696.402,Z 317.483,A -85,B 0,C 180,E1 33080.057,E2 33080.057} C_VEL
LIN {X 0,Y 696.418,Z 317.603,A -85,B 0,C 180,E1 33078.115,E2 33078.115} C_VEL
LIN {X 0,Y 697.598,Z 320.815,A -85,B 0,C 180,E1 33077.76,E2 33077.76} C_VEL
LIN {X 0,Y 698.79,Z 323.249,A -85,B 0,C 180,E1 33077.466,E2 33077.466} C_VEL
LIN {X 0,Y 705.986,Z 338.408,A -85,B 0,C 180,E1 33075.714,E2 33075.714} C_VEL
LIN {X 0,Y 708.138,Z 343.431,A -85,B 0,C 180,E1 33075.172,E2 33075.172} C_VEL
LIN {X 0,Y 708.015,Z 351.11,A -85,B 0,C 180,E1 33074.66,E2 33074.66} C_VEL
LIN {X 0,Y 712.348,Z 368.532,A -85,B 0,C 180,E1 33074.077,E2 33074.077} C_VEL
LIN {X 0,Y 710.481,Z 578.791,A -85,B 0,C 180,E1 33071.385,E2 33071.385} C_VEL
LIN {X 0,Y 708.659,Z 802.298,A -85,B 0,C 180,E1 33068.615,E2 33068.615} C_VEL
LIN {X 0,Y 708.224,Z 836.377,A -85,B 0,C 180,E1 33068.156,E2 33068.156} C_VEL
LIN {X 0,Y 707.584,Z 863.297,A -85,B 0,C 180,E1 33067.628,E2 33067.628} C_VEL
LIN {X 0,Y 706.902,Z 888.48,A -85,B 0,C 180,E1 33066.986,E2 33066.986} C_VEL
LIN {X 0,Y 705.969,Z 916.909,A -85,B 0,C 180,E1 33066.071,E2 33066.071} C_VEL
LIN {X 0,Y 705.111,Z 939.393,A -85,B 0,C 180,E1 33065.204,E2 33065.204} C_VEL
LIN {X 0,Y 704.278,Z 959.72,A -85,B 0,C 180,E1 33064.306,E2 33064.306} C_VEL
LIN {X 0,Y 703.407,Z 979.97,A -85,B 0,C 180,E1 33063.296,E2 33063.296} C_VEL
LIN {X 0,Y 702.349,Z 1004.214,A -85,B 0,C 180,E1 33061.929,E2 33061.929} C_VEL
LIN {X 0,Y 701.361,Z 1026.257,A -85,B 0,C 180,E1 33060.498,E2 33060.498} C_VEL
LIN {X 0,Y 700.54,Z 1044.723,A -85,B 0,C 180,E1 33059.166,E2 33059.166} C_VEL
LIN {X 0,Y 699.646,Z 1065.15,A -85,B 0,C 180,E1 33057.536,E2 33057.536} C_VEL
LIN {X 0,Y 698.843,Z 1084.524,A -85,B 0,C 180,E1 33055.782,E2 33055.782} C_VEL
LIN {X 0,Y 698.206,Z 1100.547,A -85,B 0,C 180,E1 33054.177,E2 33054.177} C_VEL
LIN {X 0,Y 697.593,Z 1118.362,A -85,B 0,C 180,E1 33052.189,E2 33052.189} C_VEL
LIN {X 0,Y 697.09,Z 1133.813,A -85,B 0,C 180,E1 33050.223,E2 33050.223} C_VEL
LIN {X 0,Y 696.733,Z 1146.592,A -85,B 0,C 180,E1 33048.404,E2 33048.404} C_VEL
LIN {X 0,Y 696.411,Z 1159.879,A -85,B 0,C 180,E1 33046.258,E2 33046.258} C_VEL
LIN {X 0,Y 696.216,Z 1170.714,A -85,B 0,C 180,E1 33044.205,E2 33044.205} C_VEL
LIN {X 0,Y 696.087,Z 1178.793,A -85,B 0,C 180,E1 33042.442,E2 33042.442} C_VEL
LIN {X 0,Y 695.998,Z 1186.427,A -85,B 0,C 180,E1 33040.512,E2 33040.512} C_VEL
LIN {X 0,Y 695.949,Z 1193.595,A -85,B 0,C 180,E1 33038.26,E2 33038.26} C_VEL
LIN {X 0,Y 695.92,Z 1198.937,A -85,B 0,C 180,E1 33036.02,E2 33036.02} C_VEL
LIN {X 0,Y 695.908,Z 1202.484,A -85,B 0,C 180,E1 33033.872,E2 33033.872} C_VEL
LIN {X 0,Y 695.908,Z 1204.549,A -85,B 0,C 180,E1 33031.647,E2 33031.647} C_VEL
LIN {X 0,Y 695.89,Z 1204.872,A -85,B 0,C 180,E1 33029.506,E2 33029.506} C_VEL
LIN {X 0,Y 695.907,Z 1203.961,A -85,B 0,C 180,E1 33027.53,E2 33027.53} C_VEL
LIN {X 0,Y 695.909,Z 1201.428,A -85,B 0,C 180,E1 33025.385,E2 33025.385} C_VEL
LIN {X 0,Y 695.922,Z 1197.348,A -85,B 0,C 180,E1 33023.234,E2 33023.234} C_VEL
LIN {X 0,Y 695.957,Z 1191.391,A -85,B 0,C 180,E1 33020.991,E2 33020.991} C_VEL
LIN {X 0,Y 696.017,Z 1184.162,A -85,B 0,C 180,E1 33018.871,E2 33018.871} C_VEL
LIN {X 0,Y 696.165,Z 1173.94,A -85,B 0,C 180,E1 33016.461,E2 33016.461} C_VEL
LIN {X 0,Y 696.309,Z 1164.535,A -85,B 0,C 180,E1 33014.595,E2 33014.595} C_VEL
LIN {X 0,Y 696.535,Z 1154.749,A -85,B 0,C 180,E1 33012.886,E2 33012.886} C_VEL
LIN {X 0,Y 696.81,Z 1143.682,A -85,B 0,C 180,E1 33011.164,E2 33011.164} C_VEL
LIN {X 0,Y 697.256,Z 1128.618,A -85,B 0,C 180,E1 33009.08,E2 33009.08} C_VEL
LIN {X 0,Y 697.77,Z 1112.484,A -85,B 0,C 180,E1 33007.133,E2 33007.133} C_VEL
LIN {X 0,Y 698.354,Z 1097.132,A -85,B 0,C 180,E1 33005.468,E2 33005.468} C_VEL
LIN {X 0,Y 699.102,Z 1077.878,A -85,B 0,C 180,E1 33003.59,E2 33003.59} C_VEL
LIN {X 0,Y 699.908,Z 1059.06,A -85,B 0,C 180,E1 33001.966,E2 33001.966} C_VEL
LIN {X 0,Y 700.676,Z 1041.637,A -85,B 0,C 180,E1 33000.601,E2 33000.601} C_VEL
LIN {X 0,Y 701.655,Z 1019.543,A -85,B 0,C 180,E1 32999.041,E2 32999.041} C_VEL
LIN {X 0,Y 702.662,Z 997.051,A -85,B 0,C 180,E1 32997.654,E2 32997.654} C_VEL
LIN {X 0,Y 703.513,Z 977.658,A -85,B 0,C 180,E1 32996.583,E2 32996.583} C_VEL
LIN {X 0,Y 704.372,Z 957.733,A -85,B 0,C 180,E1 32995.6,E2 32995.6} C_VEL
LIN {X 0,Y 705.354,Z 933.855,A -85,B 0,C 180,E1 32994.566,E2 32994.566} C_VEL
LIN {X 0,Y 706.253,Z 907.072,A -85,B 0,C 180,E1 32993.591,E2 32993.591} C_VEL
LIN {X 0,Y 707.026,Z 883.676,A -85,B 0,C 180,E1 32992.881,E2 32992.881} C_VEL
LIN {X 0,Y 707.751,Z 857.861,A -85,B 0,C 180,E1 32992.252,E2 32992.252} C_VEL
LIN {X 0,Y 708.321,Z 830.11,A -85,B 0,C 180,E1 32991.745,E2 32991.745} C_VEL
LIN {X 0,Y 709.322,Z 718.523,A -85,B 0,C 180,E1 32990.357,E2 32990.357} C_VEL
LIN {X 0,Y 711.206,Z 496.443,A -85,B 0,C 180,E1 32987.573,E2 32987.573} C_VEL
LIN {X 0,Y 712.225,Z 367.35,A -85,B 0,C 180,E1 32985.898,E2 32985.898} C_VEL
LIN {X 0,Y 707.901,Z 350.268,A -85,B 0,C 180,E1 32985.301,E2 32985.301} C_VEL
LIN {X 0,Y 708.077,Z 343.13,A -85,B 0,C 180,E1 32984.801,E2 32984.801} C_VEL
LIN {X 0,Y 700.067,Z 325.696,A -85,B 0,C 180,E1 32982.833,E2 32982.833} C_VEL
LIN {X 0,Y 697.597,Z 320.815,A -85,B 0,C 180,E1 32982.24,E2 32982.24} C_VEL
LIN {X 0,Y 696.4,Z 317.48,A -85,B 0,C 180,E1 32981.857,E2 32981.857} C_VEL
LIN {X 0,Y 696.378,Z 317.485,A -85,B 0,C 180,E1 32978.863,E2 32978.863} C_VEL
LIN {X 0,Y 696.401,Z 317.489,A -85,B 0,C 180,E1 32975.759,E2 32975.759} C_VEL
LIN {X 0,Y 696.37,Z 317.48,A -85,B 0,C 180,E1 32972.774,E2 32972.774} C_VEL
LIN {X 0,Y 696.404,Z 317.471,A -85,B 0,C 180,E1 32969.693,E2 32969.693} C_VEL
LIN {X 0,Y 696.358,Z 317.482,A -85,B 0,C 180,E1 32966.8,E2 32966.8} C_VEL
LIN {X 0,Y 696.399,Z 317.475,A -85,B 0,C 180,E1 32963.855,E2 32963.855} C_VEL
LIN {X 0,Y 696.353,Z 317.472,A -85,B 0,C 180,E1 32960.949,E2 32960.949} C_VEL
LIN {X 0,Y 696.393,Z 317.479,A -85,B 0,C 180,E1 32958.067,E2 32958.067} C_VEL
LIN {X 0,Y 696.357,Z 317.472,A -85,B 0,C 180,E1 32954.979,E2 32954.979} C_VEL
LIN {X 0,Y 696.355,Z 317.483,A -85,B 0,C 180,E1 32952.27,E2 32952.27} C_VEL
LIN {X 0,Y 696.396,Z 317.47,A -85,B 0,C 180,E1 32949.254,E2 32949.254} C_VEL
LIN {X 0,Y 696.338,Z 317.486,A -85,B 0,C 180,E1 32946.431,E2 32946.431} C_VEL
LIN {X 0,Y 696.397,Z 317.473,A -85,B 0,C 180,E1 32943.622,E2 32943.622} C_VEL
LIN {X 0,Y 696.347,Z 317.488,A -85,B 0,C 180,E1 32940.658,E2 32940.658} C_VEL
LIN {X 0,Y 696.336,Z 317.477,A -85,B 0,C 180,E1 32938.025,E2 32938.025} C_VEL
LIN {X 0,Y 696.401,Z 317.481,A -85,B 0,C 180,E1 32935.058,E2 32935.058} C_VEL
LIN {X 0,Y 696.328,Z 317.479,A -85,B 0,C 180,E1 32932.209,E2 32932.209} C_VEL
LIN {X 0,Y 696.35,Z 317.477,A -85,B 0,C 180,E1 32929.576,E2 32929.576} C_VEL
LIN {X 0,Y 696.341,Z 317.479,A -85,B 0,C 180,E1 32926.43,E2 32926.43} C_VEL
LIN {X 0,Y 696.317,Z 317.482,A -85,B 0,C 180,E1 32923.869,E2 32923.869} C_VEL
LIN {X 0,Y 696.378,Z 317.486,A -85,B 0,C 180,E1 32921.118,E2 32921.118} C_VEL
LIN {X 0,Y 696.327,Z 317.488,A -85,B 0,C 180,E1 32918.166,E2 32918.166} C_VEL
LIN {X 0,Y 696.309,Z 317.486,A -85,B 0,C 180,E1 32915.752,E2 32915.752} C_VEL
LIN {X 0,Y 696.343,Z 317.485,A -85,B 0,C 180,E1 32915.171,E2 32915.171} C_VEL
LIN {X 0,Y 695.419,Z 317.608,A -85,B 0,C 180,E1 32914.537,E2 32914.537} C_VEL
LIN {X 0,Y 688.891,Z 318.427,A -85,B 0,C 180,E1 32912.716,E2 32912.716} C_VEL
LIN {X 0,Y 688.411,Z 318.48,A -85,B 0,C 180,E1 32912.3,E2 32912.3} C_VEL
LIN {X 0,Y 688.364,Z 318.462,A -85,B 0,C 180,E1 32909.732,E2 32909.732} C_VEL
LIN {X 0,Y 688.37,Z 318.481,A -85,B 0,C 180,E1 32907.292,E2 32907.292} C_VEL
LIN {X 0,Y 688.442,Z 318.467,A -85,B 0,C 180,E1 32904.38,E2 32904.38} C_VEL
LIN {X 0,Y 688.355,Z 318.466,A -85,B 0,C 180,E1 32901.559,E2 32901.559} C_VEL
LIN {X 0,Y 688.358,Z 318.484,A -85,B 0,C 180,E1 32899.18,E2 32899.18} C_VEL
LIN {X 0,Y 688.446,Z 318.561,A -85,B 0,C 180,E1 32896.445,E2 32896.445} C_VEL
LIN {X 0,Y 689.515,Z 321.61,A -85,B 0,C 180,E1 32896.147,E2 32896.147} C_VEL
LIN {X 0,Y 701.237,Z 338.609,A -85,B 0,C 180,E1 32894.916,E2 32894.916} C_VEL
LIN {X 0,Y 706.451,Z 346.771,A -85,B 0,C 180,E1 32894.382,E2 32894.382} C_VEL
LIN {X 0,Y 704.535,Z 542.968,A -85,B 0,C 180,E1 32891.845,E2 32891.845} C_VEL
LIN {X 0,Y 702.427,Z 769.508,A -85,B 0,C 180,E1 32889.013,E2 32889.013} C_VEL
LIN {X 0,Y 701.926,Z 805.799,A -85,B 0,C 180,E1 32888.527,E2 32888.527} C_VEL
LIN {X 0,Y 701.216,Z 832.93,A -85,B 0,C 180,E1 32887.994,E2 32887.994} C_VEL
LIN {X 0,Y 700.448,Z 857.491,A -85,B 0,C 180,E1 32887.368,E2 32887.368} C_VEL
LIN {X 0,Y 699.459,Z 885.064,A -85,B 0,C 180,E1 32886.488,E2 32886.488} C_VEL
LIN {X 0,Y 698.432,Z 908.919,A -85,B 0,C 180,E1 32885.568,E2 32885.568} C_VEL
LIN {X 0,Y 697.518,Z 928.831,A -85,B 0,C 180,E1 32884.686,E2 32884.686} C_VEL
LIN {X 0,Y 696.555,Z 948.632,A -85,B 0,C 180,E1 32883.696,E2 32883.696} C_VEL
LIN {X 0,Y 695.56,Z 968.722,A -85,B 0,C 180,E1 32882.571,E2 32882.571} C_VEL
LIN {X 0,Y 694.273,Z 993.628,A -85,B 0,C 180,E1 32880.988,E2 32880.988} C_VEL
LIN {X 0,Y 693.291,Z 1013.151,A -85,B 0,C 180,E1 32879.579,E2 32879.579} C_VEL
LIN {X 0,Y 692.429,Z 1030.744,A -85,B 0,C 180,E1 32878.176,E2 32878.176} C_VEL
LIN {X 0,Y 691.417,Z 1051.276,A -85,B 0,C 180,E1 32876.356,E2 32876.356} C_VEL
LIN {X 0,Y 690.65,Z 1068.753,A -85,B 0,C 180,E1 32874.606,E2 32874.606} C_VEL
LIN {X 0,Y 689.968,Z 1084.796,A -85,B 0,C 180,E1 32872.826,E2 32872.826} C_VEL
LIN {X 0,Y 689.326,Z 1101.935,A -85,B 0,C 180,E1 32870.675,E2 32870.675} C_VEL
LIN {X 0,Y 688.926,Z 1114.695,A -85,B 0,C 180,E1 32868.862,E2 32868.862} C_VEL
LIN {X 0,Y 688.6,Z 1126.048,A -85,B 0,C 180,E1 32867.056,E2 32867.056} C_VEL
LIN {X 0,Y 688.313,Z 1138.393,A -85,B 0,C 180,E1 32864.813,E2 32864.813} C_VEL
LIN {X 0,Y 688.136,Z 1148.248,A -85,B 0,C 180,E1 32862.674,E2 32862.674} C_VEL
LIN {X 0,Y 688.008,Z 1155.964,A -85,B 0,C 180,E1 32860.72,E2 32860.72} C_VEL
LIN {X 0,Y 687.963,Z 1163.224,A -85,B 0,C 180,E1 32858.441,E2 32858.441} C_VEL
LIN {X 0,Y 687.931,Z 1168.673,A -85,B 0,C 180,E1 32856.174,E2 32856.174} C_VEL
LIN {X 0,Y 687.916,Z 1172.315,A -85,B 0,C 180,E1 32854.001,E2 32854.001} C_VEL
LIN {X 0,Y 687.907,Z 1174.463,A -85,B 0,C 180,E1 32851.749,E2 32851.749} C_VEL
LIN {X 0,Y 687.891,Z 1174.884,A -85,B 0,C 180,E1 32849.5,E2 32849.5} C_VEL
LIN {X 0,Y 687.906,Z 1173.995,A -85,B 0,C 180,E1 32847.501,E2 32847.501} C_VEL
LIN {X 0,Y 687.909,Z 1171.496,A -85,B 0,C 180,E1 32845.331,E2 32845.331} C_VEL
LIN {X 0,Y 687.925,Z 1167.301,A -85,B 0,C 180,E1 32843.09,E2 32843.09} C_VEL
LIN {X 0,Y 687.967,Z 1161.523,A -85,B 0,C 180,E1 32840.885,E2 32840.885} C_VEL
LIN {X 0,Y 688.038,Z 1154.447,A -85,B 0,C 180,E1 32838.771,E2 32838.771} C_VEL
LIN {X 0,Y 688.193,Z 1144.151,A -85,B 0,C 180,E1 32836.301,E2 32836.301} C_VEL
LIN {X 0,Y 688.396,Z 1134.311,A -85,B 0,C 180,E1 32834.327,E2 32834.327} C_VEL
LIN {X 0,Y 688.634,Z 1124.199,A -85,B 0,C 180,E1 32832.547,E2 32832.547} C_VEL
LIN {X 0,Y 689.016,Z 1111.65,A -85,B 0,C 180,E1 32830.591,E2 32830.591} C_VEL
LIN {X 0,Y 689.563,Z 1095.466,A -85,B 0,C 180,E1 32828.389,E2 32828.389} C_VEL
LIN {X 0,Y 690.142,Z 1080.679,A -85,B 0,C 180,E1 32826.612,E2 32826.612} C_VEL
LIN {X 0,Y 690.875,Z 1063.285,A -85,B 0,C 180,E1 32824.727,E2 32824.727} C_VEL
LIN {X 0,Y 691.768,Z 1044.313,A -85,B 0,C 180,E1 32822.917,E2 32822.917} C_VEL
LIN {X 0,Y 692.575,Z 1027.375,A -85,B 0,C 180,E1 32821.454,E2 32821.454} C_VEL
LIN {X 0,Y 693.622,Z 1006.799,A -85,B 0,C 180,E1 32819.848,E2 32819.848} C_VEL
LIN {X 0,Y 694.76,Z 984.404,A -85,B 0,C 180,E1 32818.313,E2 32818.313} C_VEL
LIN {X 0,Y 695.729,Z 965.387,A -85,B 0,C 180,E1 32817.145,E2 32817.145} C_VEL
LIN {X 0,Y 696.702,Z 945.796,A -85,B 0,C 180,E1 32816.064,E2 32816.064} C_VEL
LIN {X 0,Y 697.769,Z 923.605,A -85,B 0,C 180,E1 32814.978,E2 32814.978} C_VEL
LIN {X 0,Y 698.879,Z 897.557,A -85,B 0,C 180,E1 32813.883,E2 32813.883} C_VEL
LIN {X 0,Y 699.795,Z 874.701,A -85,B 0,C 180,E1 32813.073,E2 32813.073} C_VEL
LIN {X 0,Y 700.639,Z 851.889,A -85,B 0,C 180,E1 32812.388,E2 32812.388} C_VEL
LIN {X 0,Y 701.47,Z 824.908,A -85,B 0,C 180,E1 32811.738,E2 32811.738} C_VEL
LIN {X 0,Y 702.071,Z 797.503,A -85,B 0,C 180,E1 32811.257,E2 32811.257} C_VEL
LIN {X 0,Y 704.257,Z 571.862,A -85,B 0,C 180,E1 32808.431,E2 32808.431} C_VEL
LIN {X 0,Y 706.302,Z 363.947,A -85,B 0,C 180,E1 32805.756,E2 32805.756} C_VEL
LIN {X 0,Y 706.276,Z 346.312,A -85,B 0,C 180,E1 32805.508,E2 32805.508} C_VEL
LIN {X 0,Y 696.491,Z 331.654,A -85,B 0,C 180,E1 32804.503,E2 32804.503} C_VEL
LIN {X 0,Y 689.053,Z 320.664,A -85,B 0,C 180,E1 32803.688,E2 32803.688} C_VEL
LIN {X 0,Y 688.431,Z 318.481,A -85,B 0,C 180,E1 32803.433,E2 32803.433} C_VEL
LIN {X 0,Y 688.364,Z 318.484,A -85,B 0,C 180,E1 32800.708,E2 32800.708} C_VEL
LIN {X 0,Y 688.364,Z 318.483,A -85,B 0,C 180,E1 32798.334,E2 32798.334} C_VEL
LIN {X 0,Y 688.447,Z 318.463,A -85,B 0,C 180,E1 32795.416,E2 32795.416} C_VEL
LIN {X 0,Y 688.357,Z 318.482,A -85,B 0,C 180,E1 32792.599,E2 32792.599} C_VEL
LIN {X 0,Y 688.358,Z 318.464,A -85,B 0,C 180,E1 32790.172,E2 32790.172} C_VEL
LIN {X 0,Y 688.453,Z 318.473,A -85,B 0,C 180,E1 32787.32,E2 32787.32} C_VEL
LIN {X 0,Y 688.366,Z 318.474,A -85,B 0,C 180,E1 32784.395,E2 32784.395} C_VEL
LIN {X 0,Y 688.369,Z 318.478,A -85,B 0,C 180,E1 32782.009,E2 32782.009} C_VEL
LIN {X 0,Y 688.458,Z 318.463,A -85,B 0,C 180,E1 32779.162,E2 32779.162} C_VEL
LIN {X 0,Y 688.377,Z 318.472,A -85,B 0,C 180,E1 32776.242,E2 32776.242} C_VEL
LIN {X 0,Y 688.378,Z 318.465,A -85,B 0,C 180,E1 32773.781,E2 32773.781} C_VEL
LIN {X 0,Y 688.465,Z 318.468,A -85,B 0,C 180,E1 32770.883,E2 32770.883} C_VEL
LIN {X 0,Y 688.385,Z 318.465,A -85,B 0,C 180,E1 32768.016,E2 32768.016} C_VEL
LIN {X 0,Y 688.394,Z 318.478,A -85,B 0,C 180,E1 32765.501,E2 32765.501} C_VEL
LIN {X 0,Y 688.448,Z 318.457,A -85,B 0,C 180,E1 32762.497,E2 32762.497} C_VEL
LIN {X 0,Y 688.392,Z 318.475,A -85,B 0,C 180,E1 32759.75,E2 32759.75} C_VEL
LIN {X 0,Y 688.422,Z 318.462,A -85,B 0,C 180,E1 32757.086,E2 32757.086} C_VEL
LIN {X 0,Y 688.42,Z 318.472,A -85,B 0,C 180,E1 32753.997,E2 32753.997} C_VEL
LIN {X 0,Y 688.401,Z 318.466,A -85,B 0,C 180,E1 32751.312,E2 32751.312} C_VEL
LIN {X 0,Y 688.467,Z 318.473,A -85,B 0,C 180,E1 32748.353,E2 32748.353} C_VEL
LIN {X 0,Y 688.405,Z 318.46,A -85,B 0,C 180,E1 32745.447,E2 32745.447} C_VEL
LIN {X 0,Y 688.458,Z 318.476,A -85,B 0,C 180,E1 32742.586,E2 32742.586} C_VEL
LIN {X 0,Y 688.419,Z 318.456,A -85,B 0,C 180,E1 32739.51,E2 32739.51} C_VEL
LIN {X 0,Y 688.432,Z 318.478,A -85,B 0,C 180,E1 32736.73,E2 32736.73} C_VEL
LIN {X 0,Y 688.447,Z 318.467,A -85,B 0,C 180,E1 32733.613,E2 32733.613} C_VEL
LIN {X 0,Y 688.428,Z 318.465,A -85,B 0,C 180,E1 32730.694,E2 32730.694} C_VEL
LIN {X 0,Y 688.463,Z 318.468,A -85,B 0,C 180,E1 32727.692,E2 32727.692} C_VEL
LIN {X 0,Y 688.424,Z 318.473,A -85,B 0,C 180,E1 32724.787,E2 32724.787} C_VEL
LIN {X 0,Y 688.457,Z 318.462,A -85,B 0,C 180,E1 32721.884,E2 32721.884} C_VEL
LIN {X 0,Y 688.431,Z 318.478,A -85,B 0,C 180,E1 32718.919,E2 32718.919} C_VEL
LIN {X 0,Y 688.449,Z 318.635,A -85,B 0,C 180,E1 32718.771,E2 32718.771} C_VEL
LIN {X 0,Y 689.726,Z 321.932,A -85,B 0,C 180,E1 32718.397,E2 32718.397} C_VEL
LIN {X 0,Y 690.781,Z 323.938,A -85,B 0,C 180,E1 32718.142,E2 32718.142} C_VEL
LIN {X 0,Y 699.769,Z 342.918,A -85,B 0,C 180,E1 32715.903,E2 32715.903} C_VEL
LIN {X 0,Y 701.713,Z 347.386,A -85,B 0,C 180,E1 32715.412,E2 32715.412} C_VEL
LIN {X 0,Y 701.706,Z 351.11,A -85,B 0,C 180,E1 32715.171,E2 32715.171} C_VEL
LIN {X 0,Y 706.568,Z 370.737,A -85,B 0,C 180,E1 32714.501,E2 32714.501} C_VEL
LIN {X 0,Y 704.453,Z 580.625,A -85,B 0,C 180,E1 32711.794,E2 32711.794} C_VEL
LIN {X 0,Y 702.386,Z 804.078,A -85,B 0,C 180,E1 32709.002,E2 32709.002} C_VEL
LIN {X 0,Y 701.888,Z 837.35,A -85,B 0,C 180,E1 32708.545,E2 32708.545} C_VEL
LIN {X 0,Y 701.187,Z 863.706,A -85,B 0,C 180,E1 32708.022,E2 32708.022} C_VEL
LIN {X 0,Y 700.414,Z 888.789,A -85,B 0,C 180,E1 32707.377,E2 32707.377} C_VEL
LIN {X 0,Y 699.407,Z 916.199,A -85,B 0,C 180,E1 32706.491,E2 32706.491} C_VEL
LIN {X 0,Y 698.458,Z 938.372,A -85,B 0,C 180,E1 32705.636,E2 32705.636} C_VEL
LIN {X 0,Y 697.527,Z 958.63,A -85,B 0,C 180,E1 32704.74,E2 32704.74} C_VEL
LIN {X 0,Y 696.561,Z 978.553,A -85,B 0,C 180,E1 32703.746,E2 32703.746} C_VEL
LIN {X 0,Y 695.55,Z 998.916,A -85,B 0,C 180,E1 32702.604,E2 32702.604} C_VEL
LIN {X 0,Y 694.272,Z 1023.709,A -85,B 0,C 180,E1 32701.027,E2 32701.027} C_VEL
LIN {X 0,Y 693.311,Z 1042.849,A -85,B 0,C 180,E1 32699.647,E2 32699.647} C_VEL
LIN {X 0,Y 692.44,Z 1060.339,A -85,B 0,C 180,E1 32698.255,E2 32698.255} C_VEL
LIN {X 0,Y 691.439,Z 1080.798,A -85,B 0,C 180,E1 32696.448,E2 32696.448} C_VEL
LIN {X 0,Y 690.683,Z 1097.987,A -85,B 0,C 180,E1 32694.731,E2 32694.731} C_VEL
LIN {X 0,Y 690.026,Z 1113.411,A -85,B 0,C 180,E1 32693.031,E2 32693.031} C_VEL
LIN {X 0,Y 689.389,Z 1130.591,A -85,B 0,C 180,E1 32690.903,E2 32690.903} C_VEL
LIN {X 0,Y 688.935,Z 1144.264,A -85,B 0,C 180,E1 32688.971,E2 32688.971} C_VEL
LIN {X 0,Y 688.611,Z 1155.646,A -85,B 0,C 180,E1 32687.167,E2 32687.167} C_VEL
LIN {X 0,Y 688.318,Z 1167.302,A -85,B 0,C 180,E1 32685.071,E2 32685.071} C_VEL
LIN {X 0,Y 688.139,Z 1177.738,A -85,B 0,C 180,E1 32682.841,E2 32682.841} C_VEL
LIN {X 0,Y 688.007,Z 1185.822,A -85,B 0,C 180,E1 32680.805,E2 32680.805} C_VEL
LIN {X 0,Y 687.962,Z 1192.866,A -85,B 0,C 180,E1 32678.609,E2 32678.609} C_VEL
LIN {X 0,Y 687.927,Z 1198.422,A -85,B 0,C 180,E1 32676.342,E2 32676.342} C_VEL
LIN {X 0,Y 687.918,Z 1202.15,A -85,B 0,C 180,E1 32674.167,E2 32674.167} C_VEL
LIN {X 0,Y 687.911,Z 1204.325,A -85,B 0,C 180,E1 32671.999,E2 32671.999} C_VEL
LIN {X 0,Y 687.891,Z 1204.894,A -85,B 0,C 180,E1 32669.584,E2 32669.584} C_VEL
LIN {X 0,Y 687.907,Z 1203.959,A -85,B 0,C 180,E1 32667.501,E2 32667.501} C_VEL
LIN {X 0,Y 687.91,Z 1201.428,A -85,B 0,C 180,E1 32665.331,E2 32665.331} C_VEL
LIN {X 0,Y 687.927,Z 1197.152,A -85,B 0,C 180,E1 32663.071,E2 32663.071} C_VEL
LIN {X 0,Y 687.967,Z 1191.388,A -85,B 0,C 180,E1 32660.885,E2 32660.885} C_VEL
LIN {X 0,Y 688.039,Z 1184.277,A -85,B 0,C 180,E1 32658.771,E2 32658.771} C_VEL
LIN {X 0,Y 688.2,Z 1173.939,A -85,B 0,C 180,E1 32656.301,E2 32656.301} C_VEL
LIN {X 0,Y 688.395,Z 1164.292,A -85,B 0,C 180,E1 32654.368,E2 32654.368} C_VEL
LIN {X 0,Y 688.644,Z 1154.228,A -85,B 0,C 180,E1 32652.597,E2 32652.597} C_VEL
LIN {X 0,Y 688.983,Z 1142.519,A -85,B 0,C 180,E1 32650.766,E2 32650.766} C_VEL
LIN {X 0,Y 689.531,Z 1126.514,A -85,B 0,C 180,E1 32648.567,E2 32648.567} C_VEL
LIN {X 0,Y 690.12,Z 1111.233,A -85,B 0,C 180,E1 32646.72,E2 32646.72} C_VEL
LIN {X 0,Y 690.811,Z 1094.573,A -85,B 0,C 180,E1 32644.908,E2 32644.908} C_VEL
LIN {X 0,Y 691.75,Z 1074.837,A -85,B 0,C 180,E1 32643.009,E2 32643.009} C_VEL
LIN {X 0,Y 692.543,Z 1057.953,A -85,B 0,C 180,E1 32641.547,E2 32641.547} C_VEL
LIN {X 0,Y 693.498,Z 1038.972,A -85,B 0,C 180,E1 32640.058,E2 32640.058} C_VEL
LIN {X 0,Y 694.719,Z 1015.179,A -85,B 0,C 180,E1 32638.407,E2 32638.407} C_VEL
LIN {X 0,Y 695.721,Z 995.448,A -85,B 0,C 180,E1 32637.193,E2 32637.193} C_VEL
LIN {X 0,Y 696.697,Z 975.877,A -85,B 0,C 180,E1 32636.113,E2 32636.113} C_VEL
LIN {X 0,Y 697.765,Z 953.71,A -85,B 0,C 180,E1 32635.028,E2 32635.028} C_VEL
LIN {X 0,Y 698.897,Z 927.098,A -85,B 0,C 180,E1 32633.911,E2 32633.911} C_VEL
LIN {X 0,Y 699.789,Z 904.878,A -85,B 0,C 180,E1 32633.123,E2 32633.123} C_VEL
LIN {X 0,Y 700.634,Z 881.957,A -85,B 0,C 180,E1 32632.434,E2 32632.434} C_VEL
LIN {X 0,Y 701.462,Z 855.131,A -85,B 0,C 180,E1 32631.788,E2 32631.788} C_VEL
LIN {X 0,Y 702.068,Z 827.726,A -85,B 0,C 180,E1 32631.305,E2 32631.305} C_VEL
LIN {X 0,Y 704.225,Z 604.316,A -85,B 0,C 180,E1 32628.507,E2 32628.507} C_VEL
LIN {X 0,Y 706.316,Z 395.138,A -85,B 0,C 180,E1 32625.818,E2 32625.818} C_VEL
LIN {X 0,Y 706.413,Z 369.428,A -85,B 0,C 180,E1 32625.468,E2 32625.468} C_VEL
LIN {X 0,Y 701.598,Z 350.268,A -85,B 0,C 180,E1 32624.789,E2 32624.789} C_VEL
LIN {X 0,Y 701.499,Z 346.834,A -85,B 0,C 180,E1 32624.53,E2 32624.53} C_VEL
LIN {X 0,Y 693.838,Z 330.365,A -85,B 0,C 180,E1 32622.635,E2 32622.635} C_VEL
LIN {X 0,Y 690.137,Z 322.472,A -85,B 0,C 180,E1 32621.684,E2 32621.684} C_VEL
LIN {X 0,Y 688.591,Z 319.352,A -85,B 0,C 180,E1 32621.298,E2 32621.298} C_VEL
LIN {X 0,Y 688.426,Z 318.459,A -85,B 0,C 180,E1 32621.207,E2 32621.207} C_VEL
LIN {X 0,Y 688.459,Z 318.465,A -85,B 0,C 180,E1 32618.328,E2 32618.328} C_VEL
LIN {X 0,Y 688.43,Z 318.473,A -85,B 0,C 180,E1 32615.315,E2 32615.315} C_VEL
LIN {X 0,Y 688.461,Z 318.466,A -85,B 0,C 180,E1 32612.406,E2 32612.406} C_VEL
LIN {X 0,Y 688.431,Z 318.464,A -85,B 0,C 180,E1 32609.306,E2 32609.306} C_VEL
LIN {X 0,Y 688.451,Z 318.467,A -85,B 0,C 180,E1 32606.352,E2 32606.352} C_VEL
LIN {X 0,Y 688.435,Z 318.478,A -85,B 0,C 180,E1 32603.27,E2 32603.27} C_VEL
LIN {X 0,Y 688.42,Z 318.456,A -85,B 0,C 180,E1 32600.481,E2 32600.481} C_VEL
LIN {X 0,Y 688.461,Z 318.477,A -85,B 0,C 180,E1 32597.409,E2 32597.409} C_VEL
LIN {X 0,Y 688.406,Z 318.459,A -85,B 0,C 180,E1 32594.553,E2 32594.553} C_VEL
LIN {X 0,Y 688.466,Z 318.472,A -85,B 0,C 180,E1 32591.647,E2 32591.647} C_VEL
LIN {X 0,Y 688.406,Z 318.464,A -85,B 0,C 180,E1 32588.688,E2 32588.688} C_VEL
LIN {X 0,Y 688.421,Z 318.473,A -85,B 0,C 180,E1 32586.003,E2 32586.003} C_VEL
LIN {X 0,Y 688.419,Z 318.461,A -85,B 0,C 180,E1 32582.831,E2 32582.831} C_VEL
LIN {X 0,Y 688.398,Z 318.475,A -85,B 0,C 180,E1 32580.166,E2 32580.166} C_VEL
LIN {X 0,Y 688.464,Z 318.456,A -85,B 0,C 180,E1 32577.253,E2 32577.253} C_VEL
LIN {X 0,Y 688.393,Z 318.477,A -85,B 0,C 180,E1 32574.332,E2 32574.332} C_VEL
LIN {X 0,Y 688.402,Z 318.465,A -85,B 0,C 180,E1 32571.732,E2 32571.732} C_VEL
LIN {X 0,Y 688.417,Z 318.479,A -85,B 0,C 180,E1 32568.607,E2 32568.607} C_VEL
LIN {X 0,Y 688.38,Z 318.466,A -85,B 0,C 180,E1 32565.962,E2 32565.962} C_VEL
LIN {X 0,Y 688.423,Z 318.469,A -85,B 0,C 180,E1 32563.287,E2 32563.287} C_VEL
LIN {X 0,Y 688.388,Z 318.462,A -85,B 0,C 180,E1 32560.218,E2 32560.218} C_VEL
LIN {X 0,Y 688.375,Z 318.476,A -85,B 0,C 180,E1 32557.704,E2 32557.704} C_VEL
LIN {X 0,Y 688.426,Z 318.467,A -85,B 0,C 180,E1 32554.997,E2 32554.997} C_VEL
LIN {X 0,Y 688.411,Z 318.48,A -85,B 0,C 180,E1 32552.3,E2 32552.3} C_VEL
LIN {X 0,Y 687.365,Z 318.606,A -85,B 0,C 180,E1 32551.659,E2 32551.659} C_VEL
LIN {X 0,Y 680.944,Z 319.388,A -85,B 0,C 180,E1 32549.862,E2 32549.862} C_VEL
LIN {X 0,Y 680.429,Z 319.45,A -85,B 0,C 180,E1 32549.395,E2 32549.395} C_VEL
LIN {X 0,Y 680.51,Z 319.454,A -85,B 0,C 180,E1 32546.463,E2 32546.463} C_VEL
LIN {X 0,Y 680.423,Z 319.472,A -85,B 0,C 180,E1 32543.636,E2 32543.636} C_VEL
LIN {X 0,Y 680.423,Z 319.454,A -85,B 0,C 180,E1 32541.135,E2 32541.135} C_VEL
LIN {X 0,Y 680.487,Z 319.47,A -85,B 0,C 180,E1 32538.155,E2 32538.155} C_VEL
LIN {X 0,Y 680.446,Z 319.642,A -85,B 0,C 180,E1 32537.07,E2 32537.07} C_VEL
LIN {X 0,Y 681.008,Z 321.607,A -85,B 0,C 180,E1 32536.899,E2 32536.899} C_VEL
LIN {X 0,Y 683.048,Z 324.429,A -85,B 0,C 180,E1 32536.674,E2 32536.674} C_VEL
LIN {X 0,Y 690.417,Z 334.965,A -85,B 0,C 180,E1 32535.873,E2 32535.873} C_VEL
LIN {X 0,Y 700.677,Z 350.18,A -85,B 0,C 180,E1 32534.798,E2 32534.798} C_VEL
LIN {X 0,Y 698.574,Z 542.765,A -85,B 0,C 180,E1 32532.288,E2 32532.288} C_VEL
LIN {X 0,Y 696.214,Z 769.112,A -85,B 0,C 180,E1 32529.435,E2 32529.435} C_VEL
LIN {X 0,Y 695.647,Z 806.002,A -85,B 0,C 180,E1 32528.937,E2 32528.937} C_VEL
LIN {X 0,Y 694.871,Z 832.936,A -85,B 0,C 180,E1 32528.404,E2 32528.404} C_VEL
LIN {X 0,Y 694.018,Z 857.28,A -85,B 0,C 180,E1 32527.781,E2 32527.781} C_VEL
LIN {X 0,Y 692.903,Z 885.078,A -85,B 0,C 180,E1 32526.89,E2 32526.89} C_VEL
LIN {X 0,Y 691.778,Z 908.62,A -85,B 0,C 180,E1 32525.977,E2 32525.977} C_VEL
LIN {X 0,Y 690.745,Z 928.844,A -85,B 0,C 180,E1 32525.076,E2 32525.076} C_VEL
LIN {X 0,Y 689.673,Z 948.646,A -85,B 0,C 180,E1 32524.079,E2 32524.079} C_VEL
LIN {X 0,Y 688.519,Z 969.538,A -85,B 0,C 180,E1 32522.896,E2 32522.896} C_VEL
LIN {X 0,Y 687.062,Z 994.302,A -85,B 0,C 180,E1 32521.301,E2 32521.301} C_VEL
LIN {X 0,Y 685.981,Z 1013.493,A -85,B 0,C 180,E1 32519.9,E2 32519.9} C_VEL
LIN {X 0,Y 684.979,Z 1031.858,A -85,B 0,C 180,E1 32518.415,E2 32518.415} C_VEL
LIN {X 0,Y 683.791,Z 1053.146,A -85,B 0,C 180,E1 32516.486,E2 32516.486} C_VEL
LIN {X 0,Y 682.988,Z 1069.568,A -85,B 0,C 180,E1 32514.813,E2 32514.813} C_VEL
LIN {X 0,Y 682.204,Z 1086.112,A -85,B 0,C 180,E1 32512.946,E2 32512.946} C_VEL
LIN {X 0,Y 681.504,Z 1102.562,A -85,B 0,C 180,E1 32510.836,E2 32510.836} C_VEL
LIN {X 0,Y 681.054,Z 1115.25,A -85,B 0,C 180,E1 32509.004,E2 32509.004} C_VEL
LIN {X 0,Y 680.672,Z 1127.089,A -85,B 0,C 180,E1 32507.085,E2 32507.085} C_VEL
LIN {X 0,Y 680.344,Z 1139.628,A -85,B 0,C 180,E1 32504.729,E2 32504.729} C_VEL
LIN {X 0,Y 680.161,Z 1148.608,A -85,B 0,C 180,E1 32502.739,E2 32502.739} C_VEL
LIN {X 0,Y 680.02,Z 1156.266,A -85,B 0,C 180,E1 32500.762,E2 32500.762} C_VEL
LIN {X 0,Y 679.968,Z 1163.469,A -85,B 0,C 180,E1 32498.456,E2 32498.456} C_VEL
LIN {X 0,Y 679.932,Z 1168.846,A -85,B 0,C 180,E1 32496.162,E2 32496.162} C_VEL
LIN {X 0,Y 679.915,Z 1172.427,A -85,B 0,C 180,E1 32493.963,E2 32493.963} C_VEL
LIN {X 0,Y 679.907,Z 1174.52,A -85,B 0,C 180,E1 32491.685,E2 32491.685} C_VEL
LIN {X 0,Y 679.891,Z 1174.884,A -85,B 0,C 180,E1 32489.494,E2 32489.494} C_VEL
LIN {X 0,Y 679.906,Z 1173.992,A -85,B 0,C 180,E1 32487.471,E2 32487.471} C_VEL
LIN {X 0,Y 679.91,Z 1171.495,A -85,B 0,C 180,E1 32485.276,E2 32485.276} C_VEL
LIN {X 0,Y 679.931,Z 1167.256,A -85,B 0,C 180,E1 32482.989,E2 32482.989} C_VEL
LIN {X 0,Y 679.977,Z 1161.519,A -85,B 0,C 180,E1 32480.777,E2 32480.777} C_VEL
LIN {X 0,Y 680.065,Z 1154.445,A -85,B 0,C 180,E1 32478.638,E2 32478.638} C_VEL
LIN {X 0,Y 680.224,Z 1144.553,A -85,B 0,C 180,E1 32476.224,E2 32476.224} C_VEL
LIN {X 0,Y 680.458,Z 1134.775,A -85,B 0,C 180,E1 32474.226,E2 32474.226} C_VEL
LIN {X 0,Y 680.733,Z 1124.494,A -85,B 0,C 180,E1 32472.388,E2 32472.388} C_VEL
LIN {X 0,Y 681.149,Z 1112.231,A -85,B 0,C 180,E1 32470.447,E2 32470.447} C_VEL
LIN {X 0,Y 681.782,Z 1095.841,A -85,B 0,C 180,E1 32468.18,E2 32468.18} C_VEL
LIN {X 0,Y 682.419,Z 1081.456,A -85,B 0,C 180,E1 32466.423,E2 32466.423} C_VEL
LIN {X 0,Y 683.187,Z 1064.988,A -85,B 0,C 180,E1 32464.608,E2 32464.608} C_VEL
LIN {X 0,Y 684.238,Z 1045.274,A -85,B 0,C 180,E1 32462.684,E2 32462.684} C_VEL
LIN {X 0,Y 685.165,Z 1027.921,A -85,B 0,C 180,E1 32461.165,E2 32461.165} C_VEL
LIN {X 0,Y 686.266,Z 1008.554,A -85,B 0,C 180,E1 32459.631,E2 32459.631} C_VEL
LIN {X 0,Y 687.63,Z 985.052,A -85,B 0,C 180,E1 32457.989,E2 32457.989} C_VEL
LIN {X 0,Y 688.744,Z 965.378,A -85,B 0,C 180,E1 32456.769,E2 32456.769} C_VEL
LIN {X 0,Y 689.828,Z 945.781,A -85,B 0,C 180,E1 32455.679,E2 32455.679} C_VEL
LIN {X 0,Y 691.066,Z 922.583,A -85,B 0,C 180,E1 32454.537,E2 32454.537} C_VEL
LIN {X 0,Y 692.314,Z 896.844,A -85,B 0,C 180,E1 32453.458,E2 32453.458} C_VEL
LIN {X 0,Y 693.292,Z 874.686,A -85,B 0,C 180,E1 32452.668,E2 32452.668} C_VEL
LIN {X 0,Y 694.226,Z 851.822,A -85,B 0,C 180,E1 32451.978,E2 32451.978} C_VEL
LIN {X 0,Y 695.144,Z 825.008,A -85,B 0,C 180,E1 32451.329,E2 32451.329} C_VEL
LIN {X 0,Y 695.813,Z 797.641,A -85,B 0,C 180,E1 32450.846,E2 32450.846} C_VEL
LIN {X 0,Y 698.236,Z 574.222,A -85,B 0,C 180,E1 32448.024,E2 32448.024} C_VEL
LIN {X 0,Y 700.542,Z 365.417,A -85,B 0,C 180,E1 32445.317,E2 32445.317} C_VEL
LIN {X 0,Y 700.554,Z 349.976,A -85,B 0,C 180,E1 32445.099,E2 32445.099} C_VEL
LIN {X 0,Y 686.298,Z 328.9,A -85,B 0,C 180,E1 32443.59,E2 32443.59} C_VEL
LIN {X 0,Y 683.084,Z 324.457,A -85,B 0,C 180,E1 32443.24,E2 32443.24} C_VEL
LIN {X 0,Y 680.985,Z 321.537,A -85,B 0,C 180,E1 32443.008,E2 32443.008} C_VEL
LIN {X 0,Y 680.429,Z 319.471,A -85,B 0,C 180,E1 32442.816,E2 32442.816} C_VEL
LIN {X 0,Y 680.427,Z 319.474,A -85,B 0,C 180,E1 32440.395,E2 32440.395} C_VEL
LIN {X 0,Y 680.512,Z 319.463,A -85,B 0,C 180,E1 32437.495,E2 32437.495} C_VEL
LIN {X 0,Y 680.417,Z 319.452,A -85,B 0,C 180,E1 32434.623,E2 32434.623} C_VEL
LIN {X 0,Y 680.423,Z 319.472,A -85,B 0,C 180,E1 32432.138,E2 32432.138} C_VEL
LIN {X 0,Y 680.501,Z 319.455,A -85,B 0,C 180,E1 32429.198,E2 32429.198} C_VEL
LIN {X 0,Y 680.424,Z 319.46,A -85,B 0,C 180,E1 32426.44,E2 32426.44} C_VEL
LIN {X 0,Y 680.434,Z 319.464,A -85,B 0,C 180,E1 32423.928,E2 32423.928} C_VEL
LIN {X 0,Y 680.507,Z 319.444,A -85,B 0,C 180,E1 32421.009,E2 32421.009} C_VEL
LIN {X 0,Y 680.435,Z 319.466,A -85,B 0,C 180,E1 32418.24,E2 32418.24} C_VEL
LIN {X 0,Y 680.447,Z 319.462,A -85,B 0,C 180,E1 32415.687,E2 32415.687} C_VEL
LIN {X 0,Y 680.491,Z 319.465,A -85,B 0,C 180,E1 32412.647,E2 32412.647} C_VEL
LIN {X 0,Y 680.441,Z 319.458,A -85,B 0,C 180,E1 32409.9,E2 32409.9} C_VEL
LIN {X 0,Y 680.49,Z 319.456,A -85,B 0,C 180,E1 32407.175,E2 32407.175} C_VEL
LIN {X 0,Y 680.461,Z 319.455,A -85,B 0,C 180,E1 32404.129,E2 32404.129} C_VEL
LIN {X 0,Y 680.453,Z 319.453,A -85,B 0,C 180,E1 32401.516,E2 32401.516} C_VEL
LIN {X 0,Y 680.527,Z 319.453,A -85,B 0,C 180,E1 32398.569,E2 32398.569} C_VEL
LIN {X 0,Y 680.458,Z 319.451,A -85,B 0,C 180,E1 32395.702,E2 32395.702} C_VEL
LIN {X 0,Y 680.488,Z 319.467,A -85,B 0,C 180,E1 32392.995,E2 32392.995} C_VEL
LIN {X 0,Y 680.479,Z 319.452,A -85,B 0,C 180,E1 32389.844,E2 32389.844} C_VEL
LIN {X 0,Y 680.474,Z 319.465,A -85,B 0,C 180,E1 32387.094,E2 32387.094} C_VEL
LIN {X 0,Y 680.521,Z 319.454,A -85,B 0,C 180,E1 32384.052,E2 32384.052} C_VEL
LIN {X 0,Y 680.469,Z 319.462,A -85,B 0,C 180,E1 32381.228,E2 32381.228} C_VEL
LIN {X 0,Y 680.526,Z 319.454,A -85,B 0,C 180,E1 32378.359,E2 32378.359} C_VEL
LIN {X 0,Y 680.48,Z 319.451,A -85,B 0,C 180,E1 32375.335,E2 32375.335} C_VEL
LIN {X 0,Y 680.517,Z 319.466,A -85,B 0,C 180,E1 32372.43,E2 32372.43} C_VEL
LIN {X 0,Y 680.495,Z 319.455,A -85,B 0,C 180,E1 32369.345,E2 32369.345} C_VEL
LIN {X 0,Y 680.513,Z 319.447,A -85,B 0,C 180,E1 32366.363,E2 32366.363} C_VEL
LIN {X 0,Y 680.501,Z 319.454,A -85,B 0,C 180,E1 32363.203,E2 32363.203} C_VEL
LIN {X 0,Y 680.525,Z 319.46,A -85,B 0,C 180,E1 32360.162,E2 32360.162} C_VEL
LIN {X 0,Y 680.55,Z 319.625,A -85,B 0,C 180,E1 32359.426,E2 32359.426} C_VEL
LIN {X 0,Y 681.826,Z 322.98,A -85,B 0,C 180,E1 32359.041,E2 32359.041} C_VEL
LIN {X 0,Y 687.301,Z 334.265,A -85,B 0,C 180,E1 32357.656,E2 32357.656} C_VEL
LIN {X 0,Y 695.141,Z 350.998,A -85,B 0,C 180,E1 32355.72,E2 32355.72} C_VEL
LIN {X 0,Y 696.226,Z 354.067,A -85,B 0,C 180,E1 32355.584,E2 32355.584} C_VEL
LIN {X 0,Y 700.829,Z 372.827,A -85,B 0,C 180,E1 32354.935,E2 32354.935} C_VEL
LIN {X 0,Y 698.465,Z 582.177,A -85,B 0,C 180,E1 32352.213,E2 32352.213} C_VEL
LIN {X 0,Y 696.148,Z 805.6,A -85,B 0,C 180,E1 32349.399,E2 32349.399} C_VEL
LIN {X 0,Y 695.581,Z 838.478,A -85,B 0,C 180,E1 32348.938,E2 32348.938} C_VEL
LIN {X 0,Y 694.821,Z 864.195,A -85,B 0,C 180,E1 32348.42,E2 32348.42} C_VEL
LIN {X 0,Y 693.947,Z 889.414,A -85,B 0,C 180,E1 32347.766,E2 32347.766} C_VEL
LIN {X 0,Y 692.784,Z 917.48,A -85,B 0,C 180,E1 32346.846,E2 32346.846} C_VEL
LIN {X 0,Y 691.79,Z 938.369,A -85,B 0,C 180,E1 32346.032,E2 32346.032} C_VEL
LIN {X 0,Y 690.755,Z 958.667,A -85,B 0,C 180,E1 32345.129,E2 32345.129} C_VEL
LIN {X 0,Y 689.673,Z 978.672,A -85,B 0,C 180,E1 32344.122,E2 32344.122} C_VEL
LIN {X 0,Y 688.5,Z 999.88,A -85,B 0,C 180,E1 32342.921,E2 32342.921} C_VEL
LIN {X 0,Y 687.043,Z 1024.7,A -85,B 0,C 180,E1 32341.318,E2 32341.318} C_VEL
LIN {X 0,Y 685.991,Z 1043.455,A -85,B 0,C 180,E1 32339.947,E2 32339.947} C_VEL
LIN {X 0,Y 684.974,Z 1061.828,A -85,B 0,C 180,E1 32338.463,E2 32338.463} C_VEL
LIN {X 0,Y 683.766,Z 1083.483,A -85,B 0,C 180,E1 32336.498,E2 32336.498} C_VEL
LIN {X 0,Y 682.984,Z 1099.696,A -85,B 0,C 180,E1 32334.844,E2 32334.844} C_VEL
LIN {X 0,Y 682.192,Z 1116.492,A -85,B 0,C 180,E1 32332.946,E2 32332.946} C_VEL
LIN {X 0,Y 681.497,Z 1132.897,A -85,B 0,C 180,E1 32330.835,E2 32330.835} C_VEL
LIN {X 0,Y 681.037,Z 1145.572,A -85,B 0,C 180,E1 32329,E2 32329} C_VEL
LIN {X 0,Y 680.643,Z 1157.899,A -85,B 0,C 180,E1 32326.991,E2 32326.991} C_VEL
LIN {X 0,Y 680.337,Z 1169.84,A -85,B 0,C 180,E1 32324.729,E2 32324.729} C_VEL
LIN {X 0,Y 680.158,Z 1178.438,A -85,B 0,C 180,E1 32322.825,E2 32322.825} C_VEL
LIN {X 0,Y 680.019,Z 1186.223,A -85,B 0,C 180,E1 32320.819,E2 32320.819} C_VEL
LIN {X 0,Y 679.964,Z 1193.354,A -85,B 0,C 180,E1 32318.541,E2 32318.541} C_VEL
LIN {X 0,Y 679.926,Z 1198.83,A -85,B 0,C 180,E1 32316.216,E2 32316.216} C_VEL
LIN {X 0,Y 679.913,Z 1202.374,A -85,B 0,C 180,E1 32314.048,E2 32314.048} C_VEL
LIN {X 0,Y 679.907,Z 1204.494,A -85,B 0,C 180,E1 32311.77,E2 32311.77} C_VEL
LIN {X 0,Y 679.891,Z 1204.872,A -85,B 0,C 180,E1 32309.494,E2 32309.494} C_VEL
LIN {X 0,Y 679.907,Z 1203.956,A -85,B 0,C 180,E1 32307.471,E2 32307.471} C_VEL
LIN {X 0,Y 679.911,Z 1201.428,A -85,B 0,C 180,E1 32305.276,E2 32305.276} C_VEL
LIN {X 0,Y 679.934,Z 1197.152,A -85,B 0,C 180,E1 32302.989,E2 32302.989} C_VEL
LIN {X 0,Y 679.978,Z 1191.385,A -85,B 0,C 180,E1 32300.777,E2 32300.777} C_VEL
LIN {X 0,Y 680.067,Z 1184.278,A -85,B 0,C 180,E1 32298.638,E2 32298.638} C_VEL
LIN {X 0,Y 680.24,Z 1173.938,A -85,B 0,C 180,E1 32296.138,E2 32296.138} C_VEL
LIN {X 0,Y 680.464,Z 1164.538,A -85,B 0,C 180,E1 32294.227,E2 32294.227} C_VEL
LIN {X 0,Y 680.75,Z 1154.23,A -85,B 0,C 180,E1 32292.388,E2 32292.388} C_VEL
LIN {X 0,Y 681.15,Z 1141.939,A -85,B 0,C 180,E1 32290.447,E2 32290.447} C_VEL
LIN {X 0,Y 681.795,Z 1125.467,A -85,B 0,C 180,E1 32288.177,E2 32288.177} C_VEL
LIN {X 0,Y 682.441,Z 1111.072,A -85,B 0,C 180,E1 32286.423,E2 32286.423} C_VEL
LIN {X 0,Y 683.272,Z 1093.721,A -85,B 0,C 180,E1 32284.518,E2 32284.518} C_VEL
LIN {X 0,Y 684.268,Z 1074.724,A -85,B 0,C 180,E1 32282.679,E2 32282.679} C_VEL
LIN {X 0,Y 685.156,Z 1057.953,A -85,B 0,C 180,E1 32281.212,E2 32281.212} C_VEL
LIN {X 0,Y 686.26,Z 1038.594,A -85,B 0,C 180,E1 32279.679,E2 32279.679} C_VEL
LIN {X 0,Y 687.621,Z 1015.181,A -85,B 0,C 180,E1 32278.043,E2 32278.043} C_VEL
LIN {X 0,Y 688.734,Z 995.45,A -85,B 0,C 180,E1 32276.818,E2 32276.818} C_VEL
LIN {X 0,Y 689.843,Z 975.498,A -85,B 0,C 180,E1 32275.709,E2 32275.709} C_VEL
LIN {X 0,Y 691.118,Z 951.696,A -85,B 0,C 180,E1 32274.54,E2 32274.54} C_VEL
LIN {X 0,Y 692.334,Z 926.433,A -85,B 0,C 180,E1 32273.487,E2 32273.487} C_VEL
LIN {X 0,Y 693.316,Z 904.148,A -85,B 0,C 180,E1 32272.695,E2 32272.695} C_VEL
LIN {X 0,Y 694.253,Z 881.072,A -85,B 0,C 180,E1 32272.002,E2 32272.002} C_VEL
LIN {X 0,Y 695.165,Z 854.151,A -85,B 0,C 180,E1 32271.357,E2 32271.357} C_VEL
LIN {X 0,Y 695.824,Z 826.985,A -85,B 0,C 180,E1 32270.881,E2 32270.881} C_VEL
LIN {X 0,Y 698.219,Z 604.952,A -85,B 0,C 180,E1 32268.078,E2 32268.078} C_VEL
LIN {X 0,Y 700.556,Z 396.284,A -85,B 0,C 180,E1 32265.375,E2 32265.375} C_VEL
LIN {X 0,Y 700.679,Z 371.588,A -85,B 0,C 180,E1 32265.035,E2 32265.035} C_VEL
LIN {X 0,Y 695.295,Z 351.235,A -85,B 0,C 180,E1 32264.297,E2 32264.297} C_VEL
LIN {X 0,Y 693.169,Z 346.766,A -85,B 0,C 180,E1 32263.82,E2 32263.82} C_VEL
LIN {X 0,Y 685.845,Z 331.196,A -85,B 0,C 180,E1 32261.97,E2 32261.97} C_VEL
LIN {X 0,Y 681.808,Z 322.934,A -85,B 0,C 180,E1 32260.954,E2 32260.954} C_VEL
LIN {X 0,Y 680.524,Z 319.44,A -85,B 0,C 180,E1 32260.547,E2 32260.547} C_VEL
LIN {X 0,Y 680.494,Z 319.448,A -85,B 0,C 180,E1 32257.468,E2 32257.468} C_VEL
LIN {X 0,Y 680.519,Z 319.45,A -85,B 0,C 180,E1 32254.487,E2 32254.487} C_VEL
LIN {X 0,Y 680.497,Z 319.461,A -85,B 0,C 180,E1 32251.388,E2 32251.388} C_VEL
LIN {X 0,Y 680.511,Z 319.454,A -85,B 0,C 180,E1 32248.429,E2 32248.429} C_VEL
LIN {X 0,Y 680.496,Z 319.447,A -85,B 0,C 180,E1 32245.314,E2 32245.314} C_VEL
LIN {X 0,Y 680.492,Z 319.461,A -85,B 0,C 180,E1 32242.452,E2 32242.452} C_VEL
LIN {X 0,Y 680.504,Z 319.452,A -85,B 0,C 180,E1 32239.305,E2 32239.305} C_VEL
LIN {X 0,Y 680.476,Z 319.458,A -85,B 0,C 180,E1 32236.475,E2 32236.475} C_VEL
LIN {X 0,Y 680.526,Z 319.449,A -85,B 0,C 180,E1 32233.51,E2 32233.51} C_VEL
LIN {X 0,Y 680.465,Z 319.456,A -85,B 0,C 180,E1 32230.584,E2 32230.584} C_VEL
LIN {X 0,Y 680.523,Z 319.448,A -85,B 0,C 180,E1 32227.684,E2 32227.684} C_VEL
LIN {X 0,Y 680.469,Z 319.456,A -85,B 0,C 180,E1 32224.72,E2 32224.72} C_VEL
LIN {X 0,Y 680.469,Z 319.451,A -85,B 0,C 180,E1 32222.021,E2 32222.021} C_VEL
LIN {X 0,Y 680.507,Z 319.458,A -85,B 0,C 180,E1 32218.99,E2 32218.99} C_VEL
LIN {X 0,Y 680.451,Z 319.454,A -85,B 0,C 180,E1 32216.209,E2 32216.209} C_VEL
LIN {X 0,Y 680.508,Z 319.462,A -85,B 0,C 180,E1 32213.419,E2 32213.419} C_VEL
LIN {X 0,Y 680.456,Z 319.454,A -85,B 0,C 180,E1 32210.387,E2 32210.387} C_VEL
LIN {X 0,Y 680.45,Z 319.465,A -85,B 0,C 180,E1 32207.784,E2 32207.784} C_VEL
LIN {X 0,Y 680.52,Z 319.443,A -85,B 0,C 180,E1 32204.839,E2 32204.839} C_VEL
LIN {X 0,Y 680.441,Z 319.467,A -85,B 0,C 180,E1 32202.026,E2 32202.026} C_VEL
LIN {X 0,Y 680.443,Z 319.447,A -85,B 0,C 180,E1 32199.529,E2 32199.529} C_VEL
LIN {X 0,Y 680.498,Z 319.465,A -85,B 0,C 180,E1 32196.535,E2 32196.535} C_VEL
LIN {X 0,Y 680.432,Z 319.458,A -85,B 0,C 180,E1 32193.842,E2 32193.842} C_VEL
LIN {X 0,Y 680.442,Z 319.468,A -85,B 0,C 180,E1 32191.312,E2 32191.312} C_VEL
LIN {X 0,Y 680.429,Z 319.45,A -85,B 0,C 180,E1 32189.395,E2 32189.395} C_VEL
LIN {X 0,Y 679.473,Z 319.577,A -85,B 0,C 180,E1 32188.746,E2 32188.746} C_VEL
LIN {X 0,Y 673.116,Z 320.386,A -85,B 0,C 180,E1 32186.929,E2 32186.929} C_VEL
LIN {X 0,Y 672.568,Z 320.442,A -85,B 0,C 180,E1 32186.456,E2 32186.456} C_VEL
LIN {X 0,Y 672.483,Z 320.462,A -85,B 0,C 180,E1 32183.611,E2 32183.611} C_VEL
LIN {X 0,Y 672.484,Z 320.441,A -85,B 0,C 180,E1 32181.137,E2 32181.137} C_VEL
LIN {X 0,Y 672.545,Z 320.459,A -85,B 0,C 180,E1 32178.144,E2 32178.144} C_VEL
LIN {X 0,Y 672.527,Z 320.697,A -85,B 0,C 180,E1 32177.725,E2 32177.725} C_VEL
LIN {X 0,Y 674.005,Z 324.252,A -85,B 0,C 180,E1 32177.5,E2 32177.5} C_VEL
LIN {X 0,Y 676.452,Z 326.878,A -85,B 0,C 180,E1 32177.233,E2 32177.233} C_VEL
LIN {X 0,Y 679.083,Z 330.718,A -85,B 0,C 180,E1 32176.934,E2 32176.934} C_VEL
LIN {X 0,Y 690.088,Z 346.615,A -85,B 0,C 180,E1 32175.731,E2 32175.731} C_VEL
LIN {X 0,Y 694.963,Z 354.319,A -85,B 0,C 180,E1 32175.209,E2 32175.209} C_VEL
LIN {X 0,Y 692.553,Z 551.209,A -85,B 0,C 180,E1 32172.627,E2 32172.627} C_VEL
LIN {X 0,Y 689.934,Z 777.938,A -85,B 0,C 180,E1 32169.748,E2 32169.748} C_VEL
LIN {X 0,Y 689.294,Z 809.96,A -85,B 0,C 180,E1 32169.287,E2 32169.287} C_VEL
LIN {X 0,Y 688.483,Z 834.896,A -85,B 0,C 180,E1 32168.777,E2 32168.777} C_VEL
LIN {X 0,Y 687.51,Z 860.25,A -85,B 0,C 180,E1 32168.111,E2 32168.111} C_VEL
LIN {X 0,Y 686.243,Z 887.659,A -85,B 0,C 180,E1 32167.204,E2 32167.204} C_VEL
LIN {X 0,Y 685.146,Z 908.518,A -85,B 0,C 180,E1 32166.386,E2 32166.386} C_VEL
LIN {X 0,Y 684.002,Z 928.853,A -85,B 0,C 180,E1 32165.473,E2 32165.473} C_VEL
LIN {X 0,Y 682.826,Z 948.64,A -85,B 0,C 180,E1 32164.469,E2 32164.469} C_VEL
LIN {X 0,Y 681.499,Z 970.353,A -85,B 0,C 180,E1 32163.228,E2 32163.228} C_VEL
LIN {X 0,Y 679.881,Z 994.953,A -85,B 0,C 180,E1 32161.621,E2 32161.621} C_VEL
LIN {X 0,Y 678.683,Z 1014.107,A -85,B 0,C 180,E1 32160.206,E2 32160.206} C_VEL
LIN {X 0,Y 677.493,Z 1033.909,A -85,B 0,C 180,E1 32158.58,E2 32158.58} C_VEL
LIN {X 0,Y 676.224,Z 1054.085,A -85,B 0,C 180,E1 32156.711,E2 32156.711} C_VEL
LIN {X 0,Y 675.33,Z 1070.391,A -85,B 0,C 180,E1 32155.024,E2 32155.024} C_VEL
LIN {X 0,Y 674.393,Z 1088.37,A -85,B 0,C 180,E1 32152.95,E2 32152.95} C_VEL
LIN {X 0,Y 673.672,Z 1103.501,A -85,B 0,C 180,E1 32150.958,E2 32150.958} C_VEL
LIN {X 0,Y 673.183,Z 1115.809,A -85,B 0,C 180,E1 32149.149,E2 32149.149} C_VEL
LIN {X 0,Y 672.727,Z 1128.634,A -85,B 0,C 180,E1 32147.025,E2 32147.025} C_VEL
LIN {X 0,Y 672.38,Z 1140.453,A -85,B 0,C 180,E1 32144.731,E2 32144.731} C_VEL
LIN {X 0,Y 672.192,Z 1148.612,A -85,B 0,C 180,E1 32142.892,E2 32142.892} C_VEL
LIN {X 0,Y 672.037,Z 1156.265,A -85,B 0,C 180,E1 32140.892,E2 32140.892} C_VEL
LIN {X 0,Y 671.973,Z 1163.471,A -85,B 0,C 180,E1 32138.557,E2 32138.557} C_VEL
LIN {X 0,Y 671.934,Z 1168.847,A -85,B 0,C 180,E1 32136.236,E2 32136.236} C_VEL
LIN {X 0,Y 671.916,Z 1172.425,A -85,B 0,C 180,E1 32134.01,E2 32134.01} C_VEL
LIN {X 0,Y 671.907,Z 1174.52,A -85,B 0,C 180,E1 32131.705,E2 32131.705} C_VEL
LIN {X 0,Y 671.891,Z 1174.884,A -85,B 0,C 180,E1 32129.488,E2 32129.488} C_VEL
LIN {X 0,Y 671.906,Z 1173.989,A -85,B 0,C 180,E1 32127.441,E2 32127.441} C_VEL
LIN {X 0,Y 671.912,Z 1171.494,A -85,B 0,C 180,E1 32125.22,E2 32125.22} C_VEL
LIN {X 0,Y 671.937,Z 1167.255,A -85,B 0,C 180,E1 32122.906,E2 32122.906} C_VEL
LIN {X 0,Y 671.989,Z 1161.514,A -85,B 0,C 180,E1 32120.666,E2 32120.666} C_VEL
LIN {X 0,Y 672.092,Z 1154.444,A -85,B 0,C 180,E1 32118.501,E2 32118.501} C_VEL
LIN {X 0,Y 672.263,Z 1144.549,A -85,B 0,C 180,E1 32116.058,E2 32116.058} C_VEL
LIN {X 0,Y 672.53,Z 1134.774,A -85,B 0,C 180,E1 32114.036,E2 32114.036} C_VEL
LIN {X 0,Y 672.85,Z 1124.492,A -85,B 0,C 180,E1 32112.175,E2 32112.175} C_VEL
LIN {X 0,Y 673.287,Z 1112.811,A -85,B 0,C 180,E1 32110.3,E2 32110.3} C_VEL
LIN {X 0,Y 673.981,Z 1096.854,A -85,B 0,C 180,E1 32108.047,E2 32108.047} C_VEL
LIN {X 0,Y 674.701,Z 1082.233,A -85,B 0,C 180,E1 32106.229,E2 32106.229} C_VEL
LIN {X 0,Y 675.502,Z 1066.692,A -85,B 0,C 180,E1 32104.486,E2 32104.486} C_VEL
LIN {X 0,Y 676.721,Z 1046.186,A -85,B 0,C 180,E1 32102.441,E2 32102.441} C_VEL
LIN {X 0,Y 677.774,Z 1028.468,A -85,B 0,C 180,E1 32100.868,E2 32100.868} C_VEL
LIN {X 0,Y 678.916,Z 1010.369,A -85,B 0,C 180,E1 32099.414,E2 32099.414} C_VEL
LIN {X 0,Y 680.469,Z 986.574,A -85,B 0,C 180,E1 32097.716,E2 32097.716} C_VEL
LIN {X 0,Y 681.759,Z 965.854,A -85,B 0,C 180,E1 32096.414,E2 32096.414} C_VEL
LIN {X 0,Y 682.985,Z 945.766,A -85,B 0,C 180,E1 32095.286,E2 32095.286} C_VEL
LIN {X 0,Y 684.426,Z 921.561,A -85,B 0,C 180,E1 32094.088,E2 32094.088} C_VEL
LIN {X 0,Y 685.778,Z 896.432,A -85,B 0,C 180,E1 32093.036,E2 32093.036} C_VEL
LIN {X 0,Y 686.832,Z 874.524,A -85,B 0,C 180,E1 32092.25,E2 32092.25} C_VEL
LIN {X 0,Y 687.849,Z 851.719,A -85,B 0,C 180,E1 32091.559,E2 32091.559} C_VEL
LIN {X 0,Y 688.864,Z 824.906,A -85,B 0,C 180,E1 32090.908,E2 32090.908} C_VEL
LIN {X 0,Y 689.595,Z 797.565,A -85,B 0,C 180,E1 32090.424,E2 32090.424} C_VEL
LIN {X 0,Y 692.248,Z 576.697,A -85,B 0,C 180,E1 32087.612,E2 32087.612} C_VEL
LIN {X 0,Y 694.818,Z 367.513,A -85,B 0,C 180,E1 32084.879,E2 32084.879} C_VEL
LIN {X 0,Y 694.824,Z 353.743,A -85,B 0,C 180,E1 32084.681,E2 32084.681} C_VEL
LIN {X 0,Y 679.73,Z 331.334,A -85,B 0,C 180,E1 32083.043,E2 32083.043} C_VEL
LIN {X 0,Y 676.829,Z 327.622,A -85,B 0,C 180,E1 32082.723,E2 32082.723} C_VEL
LIN {X 0,Y 675.79,Z 325.99,A -85,B 0,C 180,E1 32082.603,E2 32082.603} C_VEL
LIN {X 0,Y 673.351,Z 323.186,A -85,B 0,C 180,E1 32082.332,E2 32082.332} C_VEL
LIN {X 0,Y 672.531,Z 320.625,A -85,B 0,C 180,E1 32082.179,E2 32082.179} C_VEL
LIN {X 0,Y 672.513,Z 320.458,A -85,B 0,C 180,E1 32079.097,E2 32079.097} C_VEL
LIN {X 0,Y 672.481,Z 320.462,A -85,B 0,C 180,E1 32076.495,E2 32076.495} C_VEL
LIN {X 0,Y 672.507,Z 320.44,A -85,B 0,C 180,E1 32073.887,E2 32073.887} C_VEL
LIN {X 0,Y 672.492,Z 320.439,A -85,B 0,C 180,E1 32070.755,E2 32070.755} C_VEL
LIN {X 0,Y 672.482,Z 320.459,A -85,B 0,C 180,E1 32068.315,E2 32068.315} C_VEL
LIN {X 0,Y 672.515,Z 320.439,A -85,B 0,C 180,E1 32065.715,E2 32065.715} C_VEL
LIN {X 0,Y 672.504,Z 320.456,A -85,B 0,C 180,E1 32062.557,E2 32062.557} C_VEL
LIN {X 0,Y 672.489,Z 320.435,A -85,B 0,C 180,E1 32060.088,E2 32060.088} C_VEL
LIN {X 0,Y 672.557,Z 320.458,A -85,B 0,C 180,E1 32057.298,E2 32057.298} C_VEL
LIN {X 0,Y 672.506,Z 320.44,A -85,B 0,C 180,E1 32054.289,E2 32054.289} C_VEL
LIN {X 0,Y 672.506,Z 320.456,A -85,B 0,C 180,E1 32051.753,E2 32051.753} C_VEL
LIN {X 0,Y 672.585,Z 320.428,A -85,B 0,C 180,E1 32048.808,E2 32048.808} C_VEL
LIN {X 0,Y 672.509,Z 320.455,A -85,B 0,C 180,E1 32045.936,E2 32045.936} C_VEL
LIN {X 0,Y 672.528,Z 320.439,A -85,B 0,C 180,E1 32043.324,E2 32043.324} C_VEL
LIN {X 0,Y 672.532,Z 320.452,A -85,B 0,C 180,E1 32040.085,E2 32040.085} C_VEL
LIN {X 0,Y 672.518,Z 320.444,A -85,B 0,C 180,E1 32037.444,E2 32037.444} C_VEL
LIN {X 0,Y 672.589,Z 320.451,A -85,B 0,C 180,E1 32034.455,E2 32034.455} C_VEL
LIN {X 0,Y 672.521,Z 320.441,A -85,B 0,C 180,E1 32031.536,E2 32031.536} C_VEL
LIN {X 0,Y 672.577,Z 320.448,A -85,B 0,C 180,E1 32028.683,E2 32028.683} C_VEL
LIN {X 0,Y 672.533,Z 320.435,A -85,B 0,C 180,E1 32025.624,E2 32025.624} C_VEL
LIN {X 0,Y 672.557,Z 320.452,A -85,B 0,C 180,E1 32022.791,E2 32022.791} C_VEL
LIN {X 0,Y 672.552,Z 320.429,A -85,B 0,C 180,E1 32019.642,E2 32019.642} C_VEL
LIN {X 0,Y 672.553,Z 320.456,A -85,B 0,C 180,E1 32016.744,E2 32016.744} C_VEL
LIN {X 0,Y 672.569,Z 320.446,A -85,B 0,C 180,E1 32013.608,E2 32013.608} C_VEL
LIN {X 0,Y 672.548,Z 320.44,A -85,B 0,C 180,E1 32010.716,E2 32010.716} C_VEL
LIN {X 0,Y 672.583,Z 320.445,A -85,B 0,C 180,E1 32007.606,E2 32007.606} C_VEL
LIN {X 0,Y 672.551,Z 320.452,A -85,B 0,C 180,E1 32004.667,E2 32004.667} C_VEL
LIN {X 0,Y 672.585,Z 320.44,A -85,B 0,C 180,E1 32001.576,E2 32001.576} C_VEL
LIN {X 0,Y 672.598,Z 320.533,A -85,B 0,C 180,E1 32000.118,E2 32000.118} C_VEL
LIN {X 0,Y 673.979,Z 324.069,A -85,B 0,C 180,E1 31999.696,E2 31999.696} C_VEL
LIN {X 0,Y 674.974,Z 326.147,A -85,B 0,C 180,E1 31999.434,E2 31999.434} C_VEL
LIN {X 0,Y 682.82,Z 342.321,A -85,B 0,C 180,E1 31997.438,E2 31997.438} C_VEL
LIN {X 0,Y 686.977,Z 351.151,A -85,B 0,C 180,E1 31996.42,E2 31996.42} C_VEL
LIN {X 0,Y 690.777,Z 357.095,A -85,B 0,C 180,E1 31996.003,E2 31996.003} C_VEL
LIN {X 0,Y 695.128,Z 375.032,A -85,B 0,C 180,E1 31995.374,E2 31995.374} C_VEL
LIN {X 0,Y 692.515,Z 583.704,A -85,B 0,C 180,E1 31992.64,E2 31992.64} C_VEL
LIN {X 0,Y 689.95,Z 806.588,A -85,B 0,C 180,E1 31989.81,E2 31989.81} C_VEL
LIN {X 0,Y 689.316,Z 839.308,A -85,B 0,C 180,E1 31989.344,E2 31989.344} C_VEL
LIN {X 0,Y 688.494,Z 864.565,A -85,B 0,C 180,E1 31988.829,E2 31988.829} C_VEL
LIN {X 0,Y 687.523,Z 889.828,A -85,B 0,C 180,E1 31988.169,E2 31988.169} C_VEL
LIN {X 0,Y 686.224,Z 918.055,A -85,B 0,C 180,E1 31987.234,E2 31987.234} C_VEL
LIN {X 0,Y 685.095,Z 939.495,A -85,B 0,C 180,E1 31986.389,E2 31986.389} C_VEL
LIN {X 0,Y 683.955,Z 959.73,A -85,B 0,C 180,E1 31985.476,E2 31985.476} C_VEL
LIN {X 0,Y 682.724,Z 980.34,A -85,B 0,C 180,E1 31984.423,E2 31984.423} C_VEL
LIN {X 0,Y 681.198,Z 1004.941,A -85,B 0,C 180,E1 31982.994,E2 31982.994} C_VEL
LIN {X 0,Y 679.763,Z 1026.922,A -85,B 0,C 180,E1 31981.527,E2 31981.527} C_VEL
LIN {X 0,Y 678.597,Z 1045.714,A -85,B 0,C 180,E1 31980.125,E2 31980.125} C_VEL
LIN {X 0,Y 677.318,Z 1066.77,A -85,B 0,C 180,E1 31978.376,E2 31978.376} C_VEL
LIN {X 0,Y 676.137,Z 1085.458,A -85,B 0,C 180,E1 31976.62,E2 31976.62} C_VEL
LIN {X 0,Y 675.285,Z 1101.394,A -85,B 0,C 180,E1 31974.96,E2 31974.96} C_VEL
LIN {X 0,Y 674.297,Z 1120.138,A -85,B 0,C 180,E1 31972.769,E2 31972.769} C_VEL
LIN {X 0,Y 673.635,Z 1134.464,A -85,B 0,C 180,E1 31970.868,E2 31970.868} C_VEL
LIN {X 0,Y 673.124,Z 1147.17,A -85,B 0,C 180,E1 31968.984,E2 31968.984} C_VEL
LIN {X 0,Y 672.639,Z 1160.814,A -85,B 0,C 180,E1 31966.672,E2 31966.672} C_VEL
LIN {X 0,Y 672.363,Z 1171.073,A -85,B 0,C 180,E1 31964.643,E2 31964.643} C_VEL
LIN {X 0,Y 672.176,Z 1179.154,A -85,B 0,C 180,E1 31962.805,E2 31962.805} C_VEL
LIN {X 0,Y 672.03,Z 1186.719,A -85,B 0,C 180,E1 31960.805,E2 31960.805} C_VEL
LIN {X 0,Y 671.97,Z 1193.595,A -85,B 0,C 180,E1 31958.557,E2 31958.557} C_VEL
LIN {X 0,Y 671.929,Z 1198.936,A -85,B 0,C 180,E1 31956.236,E2 31956.236} C_VEL
LIN {X 0,Y 671.915,Z 1202.371,A -85,B 0,C 180,E1 31954.096,E2 31954.096} C_VEL
LIN {X 0,Y 671.907,Z 1204.494,A -85,B 0,C 180,E1 31951.791,E2 31951.791} C_VEL
LIN {X 0,Y 671.891,Z 1204.872,A -85,B 0,C 180,E1 31949.488,E2 31949.488} C_VEL
LIN {X 0,Y 671.907,Z 1203.953,A -85,B 0,C 180,E1 31947.441,E2 31947.441} C_VEL
LIN {X 0,Y 671.914,Z 1201.428,A -85,B 0,C 180,E1 31945.22,E2 31945.22} C_VEL
LIN {X 0,Y 671.941,Z 1197.152,A -85,B 0,C 180,E1 31942.906,E2 31942.906} C_VEL
LIN {X 0,Y 671.991,Z 1191.382,A -85,B 0,C 180,E1 31940.666,E2 31940.666} C_VEL
LIN {X 0,Y 672.091,Z 1184.278,A -85,B 0,C 180,E1 31938.501,E2 31938.501} C_VEL
LIN {X 0,Y 672.277,Z 1174.341,A -85,B 0,C 180,E1 31936.058,E2 31936.058} C_VEL
LIN {X 0,Y 672.534,Z 1164.539,A -85,B 0,C 180,E1 31934.036,E2 31934.036} C_VEL
LIN {X 0,Y 672.865,Z 1154.232,A -85,B 0,C 180,E1 31932.175,E2 31932.175} C_VEL
LIN {X 0,Y 673.319,Z 1141.941,A -85,B 0,C 180,E1 31930.21,E2 31930.21} C_VEL
LIN {X 0,Y 674.025,Z 1125.809,A -85,B 0,C 180,E1 31927.957,E2 31927.957} C_VEL
LIN {X 0,Y 674.751,Z 1111.074,A -85,B 0,C 180,E1 31926.138,E2 31926.138} C_VEL
LIN {X 0,Y 675.713,Z 1093.722,A -85,B 0,C 180,E1 31924.213,E2 31924.213} C_VEL
LIN {X 0,Y 676.818,Z 1074.328,A -85,B 0,C 180,E1 31922.315,E2 31922.315} C_VEL
LIN {X 0,Y 677.816,Z 1057.658,A -85,B 0,C 180,E1 31920.845,E2 31920.845} C_VEL
LIN {X 0,Y 679.089,Z 1037.983,A -85,B 0,C 180,E1 31919.276,E2 31919.276} C_VEL
LIN {X 0,Y 680.588,Z 1014.456,A -85,B 0,C 180,E1 31917.623,E2 31917.623} C_VEL
LIN {X 0,Y 681.824,Z 994.651,A -85,B 0,C 180,E1 31916.387,E2 31916.387} C_VEL
LIN {X 0,Y 683.13,Z 973.171,A -85,B 0,C 180,E1 31915.193,E2 31915.193} C_VEL
LIN {X 0,Y 684.731,Z 946.23,A -85,B 0,C 180,E1 31913.9,E2 31913.9} C_VEL
LIN {X 0,Y 685.855,Z 925.015,A -85,B 0,C 180,E1 31913.027,E2 31913.027} C_VEL
LIN {X 0,Y 686.852,Z 904.075,A -85,B 0,C 180,E1 31912.28,E2 31912.28} C_VEL
LIN {X 0,Y 687.876,Z 880.997,A -85,B 0,C 180,E1 31911.584,E2 31911.584} C_VEL
LIN {X 0,Y 688.887,Z 854.068,A -85,B 0,C 180,E1 31910.936,E2 31910.936} C_VEL
LIN {X 0,Y 689.603,Z 827.166,A -85,B 0,C 180,E1 31910.463,E2 31910.463} C_VEL
LIN {X 0,Y 692.231,Z 607.497,A -85,B 0,C 180,E1 31907.666,E2 31907.666} C_VEL
LIN {X 0,Y 694.828,Z 398.362,A -85,B 0,C 180,E1 31904.937,E2 31904.937} C_VEL
LIN {X 0,Y 694.983,Z 373.766,A -85,B 0,C 180,E1 31904.596,E2 31904.596} C_VEL
LIN {X 0,Y 690.341,Z 356.111,A -85,B 0,C 180,E1 31903.945,E2 31903.945} C_VEL
LIN {X 0,Y 686.502,Z 350.268,A -85,B 0,C 180,E1 31903.505,E2 31903.505} C_VEL
LIN {X 0,Y 678.411,Z 333.039,A -85,B 0,C 180,E1 31901.435,E2 31901.435} C_VEL
LIN {X 0,Y 673.981,Z 324.058,A -85,B 0,C 180,E1 31900.303,E2 31900.303} C_VEL
LIN {X 0,Y 672.597,Z 320.528,A -85,B 0,C 180,E1 31899.882,E2 31899.882} C_VEL
LIN {X 0,Y 672.556,Z 320.44,A -85,B 0,C 180,E1 31896.887,E2 31896.887} C_VEL
LIN {X 0,Y 672.582,Z 320.432,A -85,B 0,C 180,E1 31893.78,E2 31893.78} C_VEL
LIN {X 0,Y 672.548,Z 320.445,A -85,B 0,C 180,E1 31890.859,E2 31890.859} C_VEL
LIN {X 0,Y 672.582,Z 320.449,A -85,B 0,C 180,E1 31887.827,E2 31887.827} C_VEL
LIN {X 0,Y 672.538,Z 320.437,A -85,B 0,C 180,E1 31884.882,E2 31884.882} C_VEL
LIN {X 0,Y 672.587,Z 320.451,A -85,B 0,C 180,E1 31881.91,E2 31881.91} C_VEL
LIN {X 0,Y 672.538,Z 320.452,A -85,B 0,C 180,E1 31878.912,E2 31878.912} C_VEL
LIN {X 0,Y 672.581,Z 320.444,A -85,B 0,C 180,E1 31875.964,E2 31875.964} C_VEL
LIN {X 0,Y 672.538,Z 320.455,A -85,B 0,C 180,E1 31872.886,E2 31872.886} C_VEL
LIN {X 0,Y 672.547,Z 320.442,A -85,B 0,C 180,E1 31870.104,E2 31870.104} C_VEL
LIN {X 0,Y 672.546,Z 320.456,A -85,B 0,C 180,E1 31866.917,E2 31866.917} C_VEL
LIN {X 0,Y 672.526,Z 320.441,A -85,B 0,C 180,E1 31864.178,E2 31864.178} C_VEL
LIN {X 0,Y 672.581,Z 320.447,A -85,B 0,C 180,E1 31861.107,E2 31861.107} C_VEL
LIN {X 0,Y 672.515,Z 320.443,A -85,B 0,C 180,E1 31858.296,E2 31858.296} C_VEL
LIN {X 0,Y 672.568,Z 320.439,A -85,B 0,C 180,E1 31855.481,E2 31855.481} C_VEL
LIN {X 0,Y 672.522,Z 320.445,A -85,B 0,C 180,E1 31852.482,E2 31852.482} C_VEL
LIN {X 0,Y 672.51,Z 320.443,A -85,B 0,C 180,E1 31849.896,E2 31849.896} C_VEL
LIN {X 0,Y 672.588,Z 320.446,A -85,B 0,C 180,E1 31846.94,E2 31846.94} C_VEL
LIN {X 0,Y 672.505,Z 320.449,A -85,B 0,C 180,E1 31844.123,E2 31844.123} C_VEL
LIN {X 0,Y 672.514,Z 320.455,A -85,B 0,C 180,E1 31841.537,E2 31841.537} C_VEL
LIN {X 0,Y 672.54,Z 320.444,A -85,B 0,C 180,E1 31838.455,E2 31838.455} C_VEL
LIN {X 0,Y 672.494,Z 320.452,A -85,B 0,C 180,E1 31835.772,E2 31835.772} C_VEL
LIN {X 0,Y 672.523,Z 320.445,A -85,B 0,C 180,E1 31833.129,E2 31833.129} C_VEL
LIN {X 0,Y 672.504,Z 320.437,A -85,B 0,C 180,E1 31830.028,E2 31830.028} C_VEL
LIN {X 0,Y 672.485,Z 320.46,A -85,B 0,C 180,E1 31827.537,E2 31827.537} C_VEL
LIN {X 0,Y 672.568,Z 320.442,A -85,B 0,C 180,E1 31826.456,E2 31826.456} C_VEL
LIN {X 0,Y 671.546,Z 320.56,A -85,B 0,C 180,E1 31825.8,E2 31825.8} C_VEL
LIN {X 0,Y 665.077,Z 321.386,A -85,B 0,C 180,E1 31823.961,E2 31823.961} C_VEL
LIN {X 0,Y 664.543,Z 321.451,A -85,B 0,C 180,E1 31823.482,E2 31823.482} C_VEL
LIN {X 0,Y 664.577,Z 321.43,A -85,B 0,C 180,E1 31820.788,E2 31820.788} C_VEL
LIN {X 0,Y 664.653,Z 321.651,A -85,B 0,C 180,E1 31818.438,E2 31818.438} C_VEL
LIN {X 0,Y 665.9,Z 324.881,A -85,B 0,C 180,E1 31818.264,E2 31818.264} C_VEL
LIN {X 0,Y 668.561,Z 327.847,A -85,B 0,C 180,E1 31817.96,E2 31817.96} C_VEL
LIN {X 0,Y 671.21,Z 331.77,A -85,B 0,C 180,E1 31817.646,E2 31817.646} C_VEL
LIN {X 0,Y 672.864,Z 333.892,A -85,B 0,C 180,E1 31817.457,E2 31817.457} C_VEL
LIN {X 0,Y 678.753,Z 342.023,A -85,B 0,C 180,E1 31816.793,E2 31816.793} C_VEL
LIN {X 0,Y 689.279,Z 357.807,A -85,B 0,C 180,E1 31815.636,E2 31815.636} C_VEL
LIN {X 0,Y 686.61,Z 555.407,A -85,B 0,C 180,E1 31813.027,E2 31813.027} C_VEL
LIN {X 0,Y 683.726,Z 782.557,A -85,B 0,C 180,E1 31810.121,E2 31810.121} C_VEL
LIN {X 0,Y 683.031,Z 811.429,A -85,B 0,C 180,E1 31809.688,E2 31809.688} C_VEL
LIN {X 0,Y 682.179,Z 835.554,A -85,B 0,C 180,E1 31809.186,E2 31809.186} C_VEL
LIN {X 0,Y 681.095,Z 861.238,A -85,B 0,C 180,E1 31808.504,E2 31808.504} C_VEL
LIN {X 0,Y 679.708,Z 888.378,A -85,B 0,C 180,E1 31807.594,E2 31807.594} C_VEL
LIN {X 0,Y 678.481,Z 909.66,A -85,B 0,C 180,E1 31806.749,E2 31806.749} C_VEL
LIN {X 0,Y 677.217,Z 930.147,A -85,B 0,C 180,E1 31805.817,E2 31805.817} C_VEL
LIN {X 0,Y 675.836,Z 951.345,A -85,B 0,C 180,E1 31804.721,E2 31804.721} C_VEL
LIN {X 0,Y 674.164,Z 975.752,A -85,B 0,C 180,E1 31803.281,E2 31803.281} C_VEL
LIN {X 0,Y 672.628,Z 996.984,A -85,B 0,C 180,E1 31801.85,E2 31801.85} C_VEL
LIN {X 0,Y 671.319,Z 1016.051,A -85,B 0,C 180,E1 31800.414,E2 31800.414} C_VEL
LIN {X 0,Y 669.864,Z 1037.767,A -85,B 0,C 180,E1 31798.58,E2 31798.58} C_VEL
LIN {X 0,Y 668.638,Z 1055.489,A -85,B 0,C 180,E1 31796.894,E2 31796.894} C_VEL
LIN {X 0,Y 667.674,Z 1071.218,A -85,B 0,C 180,E1 31795.239,E2 31795.239} C_VEL
LIN {X 0,Y 666.646,Z 1089.088,A -85,B 0,C 180,E1 31793.138,E2 31793.138} C_VEL
LIN {X 0,Y 665.858,Z 1104.152,A -85,B 0,C 180,E1 31791.124,E2 31791.124} C_VEL
LIN {X 0,Y 665.294,Z 1116.887,A -85,B 0,C 180,E1 31789.216,E2 31789.216} C_VEL
LIN {X 0,Y 664.747,Z 1130.585,A -85,B 0,C 180,E1 31786.876,E2 31786.876} C_VEL
LIN {X 0,Y 664.424,Z 1140.868,A -85,B 0,C 180,E1 31784.822,E2 31784.822} C_VEL
LIN {X 0,Y 664.216,Z 1148.973,A -85,B 0,C 180,E1 31782.961,E2 31782.961} C_VEL
LIN {X 0,Y 664.051,Z 1156.567,A -85,B 0,C 180,E1 31780.936,E2 31780.936} C_VEL
LIN {X 0,Y 663.978,Z 1163.472,A -85,B 0,C 180,E1 31778.661,E2 31778.661} C_VEL
LIN {X 0,Y 663.936,Z 1168.879,A -85,B 0,C 180,E1 31776.296,E2 31776.296} C_VEL
LIN {X 0,Y 663.917,Z 1172.422,A -85,B 0,C 180,E1 31774.059,E2 31774.059} C_VEL
LIN {X 0,Y 663.907,Z 1174.521,A -85,B 0,C 180,E1 31771.726,E2 31771.726} C_VEL
LIN {X 0,Y 663.891,Z 1174.883,A -85,B 0,C 180,E1 31769.482,E2 31769.482} C_VEL
LIN {X 0,Y 663.907,Z 1173.986,A -85,B 0,C 180,E1 31767.41,E2 31767.41} C_VEL
LIN {X 0,Y 663.914,Z 1171.493,A -85,B 0,C 180,E1 31765.162,E2 31765.162} C_VEL
LIN {X 0,Y 663.943,Z 1167.253,A -85,B 0,C 180,E1 31762.82,E2 31762.82} C_VEL
LIN {X 0,Y 664,Z 1161.412,A -85,B 0,C 180,E1 31760.52,E2 31760.52} C_VEL
LIN {X 0,Y 664.114,Z 1154.123,A -85,B 0,C 180,E1 31758.273,E2 31758.273} C_VEL
LIN {X 0,Y 664.327,Z 1143.992,A -85,B 0,C 180,E1 31755.766,E2 31755.766} C_VEL
LIN {X 0,Y 664.612,Z 1134.307,A -85,B 0,C 180,E1 31753.75,E2 31753.75} C_VEL
LIN {X 0,Y 664.991,Z 1123.922,A -85,B 0,C 180,E1 31751.858,E2 31751.858} C_VEL
LIN {X 0,Y 665.583,Z 1110.479,A -85,B 0,C 180,E1 31749.695,E2 31749.695} C_VEL
LIN {X 0,Y 666.345,Z 1094.745,A -85,B 0,C 180,E1 31747.503,E2 31747.503} C_VEL
LIN {X 0,Y 667.13,Z 1080.07,A -85,B 0,C 180,E1 31745.682,E2 31745.682} C_VEL
LIN {X 0,Y 668.286,Z 1061.93,A -85,B 0,C 180,E1 31743.667,E2 31743.667} C_VEL
LIN {X 0,Y 669.402,Z 1043.783,A -85,B 0,C 180,E1 31741.885,E2 31741.885} C_VEL
LIN {X 0,Y 670.613,Z 1026.241,A -85,B 0,C 180,E1 31740.33,E2 31740.33} C_VEL
LIN {X 0,Y 672.159,Z 1004.809,A -85,B 0,C 180,E1 31738.625,E2 31738.625} C_VEL
LIN {X 0,Y 673.63,Z 982.927,A -85,B 0,C 180,E1 31737.095,E2 31737.095} C_VEL
LIN {X 0,Y 675.008,Z 962.931,A -85,B 0,C 180,E1 31735.848,E2 31735.848} C_VEL
LIN {X 0,Y 676.717,Z 938.521,A -85,B 0,C 180,E1 31734.502,E2 31734.502} C_VEL
LIN {X 0,Y 678.247,Z 913.833,A -85,B 0,C 180,E1 31733.342,E2 31733.342} C_VEL
LIN {X 0,Y 679.421,Z 893.571,A -85,B 0,C 180,E1 31732.512,E2 31732.512} C_VEL
LIN {X 0,Y 680.462,Z 873.171,A -85,B 0,C 180,E1 31731.786,E2 31731.786} C_VEL
LIN {X 0,Y 681.598,Z 849.805,A -85,B 0,C 180,E1 31731.083,E2 31731.083} C_VEL
LIN {X 0,Y 682.711,Z 822.138,A -85,B 0,C 180,E1 31730.426,E2 31730.426} C_VEL
LIN {X 0,Y 683.436,Z 796.417,A -85,B 0,C 180,E1 31729.979,E2 31729.979} C_VEL
LIN {X 0,Y 686.336,Z 576.264,A -85,B 0,C 180,E1 31727.154,E2 31727.154} C_VEL
LIN {X 0,Y 689.159,Z 367.589,A -85,B 0,C 180,E1 31724.406,E2 31724.406} C_VEL
LIN {X 0,Y 689.15,Z 357.483,A -85,B 0,C 180,E1 31724.258,E2 31724.258} C_VEL
LIN {X 0,Y 675.603,Z 337.461,A -85,B 0,C 180,E1 31722.762,E2 31722.762} C_VEL
LIN {X 0,Y 672.304,Z 332.876,A -85,B 0,C 180,E1 31722.385,E2 31722.385} C_VEL
LIN {X 0,Y 669.073,Z 328.845,A -85,B 0,C 180,E1 31722.015,E2 31722.015} C_VEL
LIN {X 0,Y 667.99,Z 327.035,A -85,B 0,C 180,E1 31721.883,E2 31721.883} C_VEL
LIN {X 0,Y 665.585,Z 324.327,A -85,B 0,C 180,E1 31721.606,E2 31721.606} C_VEL
LIN {X 0,Y 664.623,Z 321.445,A -85,B 0,C 180,E1 31721.45,E2 31721.45} C_VEL
LIN {X 0,Y 664.545,Z 321.452,A -85,B 0,C 180,E1 31718.64,E2 31718.64} C_VEL
LIN {X 0,Y 664.562,Z 321.451,A -85,B 0,C 180,E1 31716.036,E2 31716.036} C_VEL
LIN {X 0,Y 664.562,Z 321.451,A -85,B 0,C 180,E1 31712.899,E2 31712.899} C_VEL
LIN {X 0,Y 664.537,Z 321.426,A -85,B 0,C 180,E1 31710.369,E2 31710.369} C_VEL
LIN {X 0,Y 664.573,Z 321.448,A -85,B 0,C 180,E1 31707.792,E2 31707.792} C_VEL
LIN {X 0,Y 664.564,Z 321.437,A -85,B 0,C 180,E1 31704.631,E2 31704.631} C_VEL
LIN {X 0,Y 664.551,Z 321.445,A -85,B 0,C 180,E1 31702.096,E2 31702.096} C_VEL
LIN {X 0,Y 664.63,Z 321.424,A -85,B 0,C 180,E1 31699.237,E2 31699.237} C_VEL
LIN {X 0,Y 664.561,Z 321.438,A -85,B 0,C 180,E1 31696.252,E2 31696.252} C_VEL
LIN {X 0,Y 664.564,Z 321.429,A -85,B 0,C 180,E1 31693.752,E2 31693.752} C_VEL
LIN {X 0,Y 664.634,Z 321.432,A -85,B 0,C 180,E1 31690.751,E2 31690.751} C_VEL
LIN {X 0,Y 664.566,Z 321.429,A -85,B 0,C 180,E1 31687.869,E2 31687.869} C_VEL
LIN {X 0,Y 664.62,Z 321.444,A -85,B 0,C 180,E1 31685.092,E2 31685.092} C_VEL
LIN {X 0,Y 664.579,Z 321.428,A -85,B 0,C 180,E1 31681.983,E2 31681.983} C_VEL
LIN {X 0,Y 664.59,Z 321.445,A -85,B 0,C 180,E1 31679.31,E2 31679.31} C_VEL
LIN {X 0,Y 664.618,Z 321.42,A -85,B 0,C 180,E1 31676.204,E2 31676.204} C_VEL
LIN {X 0,Y 664.583,Z 321.443,A -85,B 0,C 180,E1 31673.434,E2 31673.434} C_VEL
LIN {X 0,Y 664.647,Z 321.415,A -85,B 0,C 180,E1 31670.475,E2 31670.475} C_VEL
LIN {X 0,Y 664.588,Z 321.441,A -85,B 0,C 180,E1 31667.487,E2 31667.487} C_VEL
LIN {X 0,Y 664.646,Z 321.417,A -85,B 0,C 180,E1 31664.557,E2 31664.557} C_VEL
LIN {X 0,Y 664.598,Z 321.438,A -85,B 0,C 180,E1 31661.491,E2 31661.491} C_VEL
LIN {X 0,Y 664.628,Z 321.425,A -85,B 0,C 180,E1 31658.625,E2 31658.625} C_VEL
LIN {X 0,Y 664.61,Z 321.426,A -85,B 0,C 180,E1 31655.466,E2 31655.466} C_VEL
LIN {X 0,Y 664.634,Z 321.443,A -85,B 0,C 180,E1 31652.493,E2 31652.493} C_VEL
LIN {X 0,Y 664.617,Z 321.431,A -85,B 0,C 180,E1 31649.335,E2 31649.335} C_VEL
LIN {X 0,Y 664.633,Z 321.421,A -85,B 0,C 180,E1 31646.384,E2 31646.384} C_VEL
LIN {X 0,Y 664.624,Z 321.428,A -85,B 0,C 180,E1 31643.218,E2 31643.218} C_VEL
LIN {X 0,Y 664.629,Z 321.574,A -85,B 0,C 180,E1 31640.826,E2 31640.826} C_VEL
LIN {X 0,Y 665.786,Z 324.706,A -85,B 0,C 180,E1 31640.448,E2 31640.448} C_VEL
LIN {X 0,Y 666.87,Z 326.516,A -85,B 0,C 180,E1 31640.19,E2 31640.19} C_VEL
LIN {X 0,Y 676.757,Z 347.069,A -85,B 0,C 180,E1 31637.622,E2 31637.622} C_VEL
LIN {X 0,Y 678.76,Z 351.161,A -85,B 0,C 180,E1 31637.154,E2 31637.154} C_VEL
LIN {X 0,Y 685.841,Z 361.989,A -85,B 0,C 180,E1 31636.359,E2 31636.359} C_VEL
LIN {X 0,Y 689.468,Z 377.325,A -85,B 0,C 180,E1 31635.819,E2 31635.819} C_VEL
LIN {X 0,Y 686.6,Z 585.512,A -85,B 0,C 180,E1 31633.071,E2 31633.071} C_VEL
LIN {X 0,Y 683.78,Z 808.274,A -85,B 0,C 180,E1 31630.22,E2 31630.22} C_VEL
LIN {X 0,Y 683.077,Z 840.163,A -85,B 0,C 180,E1 31629.756,E2 31629.756} C_VEL
LIN {X 0,Y 682.208,Z 864.806,A -85,B 0,C 180,E1 31629.249,E2 31629.249} C_VEL
LIN {X 0,Y 681.152,Z 889.931,A -85,B 0,C 180,E1 31628.588,E2 31628.588} C_VEL
LIN {X 0,Y 679.737,Z 917.912,A -85,B 0,C 180,E1 31627.657,E2 31627.657} C_VEL
LIN {X 0,Y 678.491,Z 939.492,A -85,B 0,C 180,E1 31626.801,E2 31626.801} C_VEL
LIN {X 0,Y 677.241,Z 959.726,A -85,B 0,C 180,E1 31625.882,E2 31625.882} C_VEL
LIN {X 0,Y 675.886,Z 980.554,A -85,B 0,C 180,E1 31624.809,E2 31624.809} C_VEL
LIN {X 0,Y 674.235,Z 1004.938,A -85,B 0,C 180,E1 31623.379,E2 31623.379} C_VEL
LIN {X 0,Y 672.655,Z 1026.642,A -85,B 0,C 180,E1 31621.92,E2 31621.92} C_VEL
LIN {X 0,Y 671.37,Z 1045.271,A -85,B 0,C 180,E1 31620.52,E2 31620.52} C_VEL
LIN {X 0,Y 669.98,Z 1066.204,A -85,B 0,C 180,E1 31618.77,E2 31618.77} C_VEL
LIN {X 0,Y 668.655,Z 1085.189,A -85,B 0,C 180,E1 31616.969,E2 31616.969} C_VEL
LIN {X 0,Y 667.705,Z 1100.547,A -85,B 0,C 180,E1 31615.358,E2 31615.358} C_VEL
LIN {X 0,Y 666.72,Z 1118.009,A -85,B 0,C 180,E1 31613.323,E2 31613.323} C_VEL
LIN {X 0,Y 665.878,Z 1133.821,A -85,B 0,C 180,E1 31611.215,E2 31611.215} C_VEL
LIN {X 0,Y 665.317,Z 1146.017,A -85,B 0,C 180,E1 31609.398,E2 31609.398} C_VEL
LIN {X 0,Y 664.82,Z 1158.891,A -85,B 0,C 180,E1 31607.234,E2 31607.234} C_VEL
LIN {X 0,Y 664.423,Z 1170.664,A -85,B 0,C 180,E1 31604.912,E2 31604.912} C_VEL
LIN {X 0,Y 664.224,Z 1178.798,A -85,B 0,C 180,E1 31603.05,E2 31603.05} C_VEL
LIN {X 0,Y 664.054,Z 1186.419,A -85,B 0,C 180,E1 31601.024,E2 31601.024} C_VEL
LIN {X 0,Y 663.977,Z 1193.595,A -85,B 0,C 180,E1 31598.661,E2 31598.661} C_VEL
LIN {X 0,Y 663.932,Z 1198.968,A -85,B 0,C 180,E1 31596.293,E2 31596.293} C_VEL
LIN {X 0,Y 663.915,Z 1202.482,A -85,B 0,C 180,E1 31594.059,E2 31594.059} C_VEL
LIN {X 0,Y 663.907,Z 1204.549,A -85,B 0,C 180,E1 31591.726,E2 31591.726} C_VEL
LIN {X 0,Y 663.891,Z 1204.872,A -85,B 0,C 180,E1 31589.482,E2 31589.482} C_VEL
LIN {X 0,Y 663.908,Z 1203.95,A -85,B 0,C 180,E1 31587.41,E2 31587.41} C_VEL
LIN {X 0,Y 663.917,Z 1201.428,A -85,B 0,C 180,E1 31585.162,E2 31585.162} C_VEL
LIN {X 0,Y 663.948,Z 1197.152,A -85,B 0,C 180,E1 31582.82,E2 31582.82} C_VEL
LIN {X 0,Y 664.001,Z 1191.28,A -85,B 0,C 180,E1 31580.519,E2 31580.519} C_VEL
LIN {X 0,Y 664.109,Z 1183.959,A -85,B 0,C 180,E1 31578.273,E2 31578.273} C_VEL
LIN {X 0,Y 664.345,Z 1173.758,A -85,B 0,C 180,E1 31575.76,E2 31575.76} C_VEL
LIN {X 0,Y 664.618,Z 1164.076,A -85,B 0,C 180,E1 31573.751,E2 31573.751} C_VEL
LIN {X 0,Y 665.008,Z 1153.637,A -85,B 0,C 180,E1 31571.854,E2 31571.854} C_VEL
LIN {X 0,Y 665.631,Z 1139.568,A -85,B 0,C 180,E1 31569.605,E2 31569.605} C_VEL
LIN {X 0,Y 666.363,Z 1124.404,A -85,B 0,C 180,E1 31567.504,E2 31567.504} C_VEL
LIN {X 0,Y 667.166,Z 1109.516,A -85,B 0,C 180,E1 31565.661,E2 31565.661} C_VEL
LIN {X 0,Y 668.348,Z 1090.654,A -85,B 0,C 180,E1 31563.582,E2 31563.582} C_VEL
LIN {X 0,Y 669.435,Z 1073.313,A -85,B 0,C 180,E1 31561.886,E2 31561.886} C_VEL
LIN {X 0,Y 670.617,Z 1056.207,A -85,B 0,C 180,E1 31560.373,E2 31560.373} C_VEL
LIN {X 0,Y 672.188,Z 1034.208,A -85,B 0,C 180,E1 31558.627,E2 31558.627} C_VEL
LIN {X 0,Y 673.617,Z 1013.162,A -85,B 0,C 180,E1 31557.156,E2 31557.156} C_VEL
LIN {X 0,Y 674.999,Z 993.054,A -85,B 0,C 180,E1 31555.9,E2 31555.9} C_VEL
LIN {X 0,Y 676.708,Z 968.661,A -85,B 0,C 180,E1 31554.554,E2 31554.554} C_VEL
LIN {X 0,Y 678.238,Z 943.998,A -85,B 0,C 180,E1 31553.394,E2 31553.394} C_VEL
LIN {X 0,Y 679.403,Z 923.896,A -85,B 0,C 180,E1 31552.57,E2 31552.57} C_VEL
LIN {X 0,Y 680.471,Z 903.03,A -85,B 0,C 180,E1 31551.826,E2 31551.826} C_VEL
LIN {X 0,Y 681.603,Z 879.634,A -85,B 0,C 180,E1 31551.123,E2 31551.123} C_VEL
LIN {X 0,Y 682.719,Z 851.802,A -85,B 0,C 180,E1 31550.464,E2 31550.464} C_VEL
LIN {X 0,Y 683.44,Z 826.276,A -85,B 0,C 180,E1 31550.022,E2 31550.022} C_VEL
LIN {X 0,Y 686.307,Z 607.878,A -85,B 0,C 180,E1 31547.219,E2 31547.219} C_VEL
LIN {X 0,Y 689.162,Z 398.958,A -85,B 0,C 180,E1 31544.471,E2 31544.471} C_VEL
LIN {X 0,Y 689.328,Z 375.958,A -85,B 0,C 180,E1 31544.149,E2 31544.149} C_VEL
LIN {X 0,Y 685.409,Z 361.022,A -85,B 0,C 180,E1 31543.589,E2 31543.589} C_VEL
LIN {X 0,Y 678.216,Z 350.268,A -85,B 0,C 180,E1 31542.763,E2 31542.763} C_VEL
LIN {X 0,Y 670.144,Z 333.469,A -85,B 0,C 180,E1 31540.695,E2 31540.695} C_VEL
LIN {X 0,Y 666.172,Z 325.251,A -85,B 0,C 180,E1 31539.636,E2 31539.636} C_VEL
LIN {X 0,Y 664.721,Z 322.095,A -85,B 0,C 180,E1 31539.227,E2 31539.227} C_VEL
LIN {X 0,Y 664.614,Z 321.446,A -85,B 0,C 180,E1 31539.133,E2 31539.133} C_VEL
LIN {X 0,Y 664.641,Z 321.437,A -85,B 0,C 180,E1 31536.115,E2 31536.115} C_VEL
LIN {X 0,Y 664.606,Z 321.431,A -85,B 0,C 180,E1 31533.102,E2 31533.102} C_VEL
LIN {X 0,Y 664.645,Z 321.42,A -85,B 0,C 180,E1 31530.118,E2 31530.118} C_VEL
LIN {X 0,Y 664.608,Z 321.44,A -85,B 0,C 180,E1 31527.12,E2 31527.12} C_VEL
LIN {X 0,Y 664.645,Z 321.423,A -85,B 0,C 180,E1 31524.155,E2 31524.155} C_VEL
LIN {X 0,Y 664.604,Z 321.424,A -85,B 0,C 180,E1 31521.074,E2 31521.074} C_VEL
LIN {X 0,Y 664.629,Z 321.435,A -85,B 0,C 180,E1 31518.145,E2 31518.145} C_VEL
LIN {X 0,Y 664.602,Z 321.419,A -85,B 0,C 180,E1 31514.997,E2 31514.997} C_VEL
LIN {X 0,Y 664.61,Z 321.439,A -85,B 0,C 180,E1 31512.159,E2 31512.159} C_VEL
LIN {X 0,Y 664.611,Z 321.419,A -85,B 0,C 180,E1 31509.002,E2 31509.002} C_VEL
LIN {X 0,Y 664.59,Z 321.442,A -85,B 0,C 180,E1 31506.219,E2 31506.219} C_VEL
LIN {X 0,Y 664.64,Z 321.415,A -85,B 0,C 180,E1 31503.191,E2 31503.191} C_VEL
LIN {X 0,Y 664.58,Z 321.443,A -85,B 0,C 180,E1 31500.345,E2 31500.345} C_VEL
LIN {X 0,Y 664.632,Z 321.419,A -85,B 0,C 180,E1 31497.499,E2 31497.499} C_VEL
LIN {X 0,Y 664.583,Z 321.445,A -85,B 0,C 180,E1 31494.474,E2 31494.474} C_VEL
LIN {X 0,Y 664.577,Z 321.43,A -85,B 0,C 180,E1 31491.869,E2 31491.869} C_VEL
LIN {X 0,Y 664.626,Z 321.44,A -85,B 0,C 180,E1 31488.809,E2 31488.809} C_VEL
LIN {X 0,Y 664.565,Z 321.43,A -85,B 0,C 180,E1 31486.029,E2 31486.029} C_VEL
LIN {X 0,Y 664.593,Z 321.435,A -85,B 0,C 180,E1 31483.39,E2 31483.39} C_VEL
LIN {X 0,Y 664.579,Z 321.424,A -85,B 0,C 180,E1 31480.305,E2 31480.305} C_VEL
LIN {X 0,Y 664.56,Z 321.443,A -85,B 0,C 180,E1 31477.712,E2 31477.712} C_VEL
LIN {X 0,Y 664.623,Z 321.424,A -85,B 0,C 180,E1 31474.896,E2 31474.896} C_VEL
LIN {X 0,Y 664.558,Z 321.448,A -85,B 0,C 180,E1 31471.905,E2 31471.905} C_VEL
LIN {X 0,Y 664.551,Z 321.424,A -85,B 0,C 180,E1 31469.432,E2 31469.432} C_VEL
LIN {X 0,Y 664.631,Z 321.43,A -85,B 0,C 180,E1 31466.487,E2 31466.487} C_VEL
LIN {X 0,Y 664.545,Z 321.451,A -85,B 0,C 180,E1 31463.605,E2 31463.605} C_VEL
LIN {X 0,Y 664.543,Z 321.451,A -85,B 0,C 180,E1 31463.482,E2 31463.482} C_VEL
LIN {X 0,Y 663.543,Z 321.573,A -85,B 0,C 180,E1 31462.818,E2 31462.818} C_VEL
LIN {X 0,Y 657.246,Z 322.34,A -85,B 0,C 180,E1 31461.005,E2 31461.005} C_VEL
LIN {X 0,Y 656.688,Z 322.418,A -85,B 0,C 180,E1 31460.473,E2 31460.473} C_VEL
LIN {X 0,Y 656.625,Z 322.61,A -85,B 0,C 180,E1 31459.226,E2 31459.226} C_VEL
LIN {X 0,Y 657.8,Z 325.745,A -85,B 0,C 180,E1 31459.055,E2 31459.055} C_VEL
LIN {X 0,Y 660.781,Z 328.871,A -85,B 0,C 180,E1 31458.704,E2 31458.704} C_VEL
LIN {X 0,Y 663.475,Z 332.863,A -85,B 0,C 180,E1 31458.373,E2 31458.373} C_VEL
LIN {X 0,Y 665.013,Z 334.863,A -85,B 0,C 180,E1 31458.191,E2 31458.191} C_VEL
LIN {X 0,Y 674.41,Z 347.67,A -85,B 0,C 180,E1 31457.101,E2 31457.101} C_VEL
LIN {X 0,Y 683.629,Z 361.611,A -85,B 0,C 180,E1 31456.067,E2 31456.067} C_VEL
LIN {X 0,Y 680.695,Z 559.955,A -85,B 0,C 180,E1 31453.429,E2 31453.429} C_VEL
LIN {X 0,Y 677.521,Z 787.726,A -85,B 0,C 180,E1 31450.491,E2 31450.491} C_VEL
LIN {X 0,Y 676.769,Z 813.76,A -85,B 0,C 180,E1 31450.08,E2 31450.08} C_VEL
LIN {X 0,Y 675.847,Z 837.73,A -85,B 0,C 180,E1 31449.568,E2 31449.568} C_VEL
LIN {X 0,Y 674.589,Z 864.786,A -85,B 0,C 180,E1 31448.826,E2 31448.826} C_VEL
LIN {X 0,Y 673.213,Z 888.969,A -85,B 0,C 180,E1 31447.997,E2 31447.997} C_VEL
LIN {X 0,Y 671.91,Z 909.671,A -85,B 0,C 180,E1 31447.168,E2 31447.168} C_VEL
LIN {X 0,Y 670.492,Z 930.881,A -85,B 0,C 180,E1 31446.194,E2 31446.194} C_VEL
LIN {X 0,Y 668.863,Z 954.028,A -85,B 0,C 180,E1 31444.979,E2 31444.979} C_VEL
LIN {X 0,Y 666.964,Z 978.696,A -85,B 0,C 180,E1 31443.482,E2 31443.482} C_VEL
LIN {X 0,Y 665.439,Z 998.325,A -85,B 0,C 180,E1 31442.134,E2 31442.134} C_VEL
LIN {X 0,Y 663.897,Z 1019.021,A -85,B 0,C 180,E1 31440.545,E2 31440.545} C_VEL
LIN {X 0,Y 662.292,Z 1040.312,A -85,B 0,C 180,E1 31438.691,E2 31438.691} C_VEL
LIN {X 0,Y 661.059,Z 1056.889,A -85,B 0,C 180,E1 31437.082,E2 31437.082} C_VEL
LIN {X 0,Y 659.91,Z 1074.374,A -85,B 0,C 180,E1 31435.198,E2 31435.198} C_VEL
LIN {X 0,Y 658.771,Z 1091.936,A -85,B 0,C 180,E1 31433.053,E2 31433.053} C_VEL
LIN {X 0,Y 658.013,Z 1105.448,A -85,B 0,C 180,E1 31431.201,E2 31431.201} C_VEL
LIN {X 0,Y 657.327,Z 1119.755,A -85,B 0,C 180,E1 31428.997,E2 31428.997} C_VEL
LIN {X 0,Y 656.761,Z 1132.451,A -85,B 0,C 180,E1 31426.722,E2 31426.722} C_VEL
LIN {X 0,Y 656.46,Z 1141.692,A -85,B 0,C 180,E1 31424.826,E2 31424.826} C_VEL
LIN {X 0,Y 656.238,Z 1149.691,A -85,B 0,C 180,E1 31422.942,E2 31422.942} C_VEL
LIN {X 0,Y 656.055,Z 1157.45,A -85,B 0,C 180,E1 31420.804,E2 31420.804} C_VEL
LIN {X 0,Y 655.98,Z 1164.382,A -85,B 0,C 180,E1 31418.406,E2 31418.406} C_VEL
LIN {X 0,Y 655.934,Z 1169.328,A -85,B 0,C 180,E1 31416.125,E2 31416.125} C_VEL
LIN {X 0,Y 655.913,Z 1172.736,A -85,B 0,C 180,E1 31413.846,E2 31413.846} C_VEL
LIN {X 0,Y 655.909,Z 1174.612,A -85,B 0,C 180,E1 31411.485,E2 31411.485} C_VEL
LIN {X 0,Y 655.893,Z 1174.861,A -85,B 0,C 180,E1 31409.389,E2 31409.389} C_VEL
LIN {X 0,Y 655.909,Z 1173.914,A -85,B 0,C 180,E1 31407.291,E2 31407.291} C_VEL
LIN {X 0,Y 655.92,Z 1171.367,A -85,B 0,C 180,E1 31405.015,E2 31405.015} C_VEL
LIN {X 0,Y 655.947,Z 1167.056,A -85,B 0,C 180,E1 31402.644,E2 31402.644} C_VEL
LIN {X 0,Y 656.009,Z 1161.251,A -85,B 0,C 180,E1 31400.348,E2 31400.348} C_VEL
LIN {X 0,Y 656.135,Z 1153.868,A -85,B 0,C 180,E1 31398.057,E2 31398.057} C_VEL
LIN {X 0,Y 656.4,Z 1143.731,A -85,B 0,C 180,E1 31395.534,E2 31395.534} C_VEL
LIN {X 0,Y 656.692,Z 1134.305,A -85,B 0,C 180,E1 31393.549,E2 31393.549} C_VEL
LIN {X 0,Y 657.105,Z 1123.966,A -85,B 0,C 180,E1 31391.641,E2 31391.641} C_VEL
LIN {X 0,Y 657.775,Z 1110.477,A -85,B 0,C 180,E1 31389.443,E2 31389.443} C_VEL
LIN {X 0,Y 658.618,Z 1094.738,A -85,B 0,C 180,E1 31387.225,E2 31387.225} C_VEL
LIN {X 0,Y 659.456,Z 1080.666,A -85,B 0,C 180,E1 31385.453,E2 31385.453} C_VEL
LIN {X 0,Y 660.703,Z 1062.795,A -85,B 0,C 180,E1 31383.433,E2 31383.433} C_VEL
LIN {X 0,Y 662.014,Z 1043.619,A -85,B 0,C 180,E1 31381.527,E2 31381.527} C_VEL
LIN {X 0,Y 663.288,Z 1026.788,A -85,B 0,C 180,E1 31380.019,E2 31380.019} C_VEL
LIN {X 0,Y 664.969,Z 1005.527,A -85,B 0,C 180,E1 31378.302,E2 31378.302} C_VEL
LIN {X 0,Y 666.624,Z 982.919,A -85,B 0,C 180,E1 31376.705,E2 31376.705} C_VEL
LIN {X 0,Y 668.141,Z 962.918,A -85,B 0,C 180,E1 31375.447,E2 31375.447} C_VEL
LIN {X 0,Y 670.008,Z 938.52,A -85,B 0,C 180,E1 31374.093,E2 31374.093} C_VEL
